LIN {X 0,Y 421.237,Z 718.592,A -85,B 0,C 180,E1 -10154.642,E2 -10154.642} C_VEL
LIN {X 0,Y 420.431,Z 729.964,A -85,B 0,C 180,E1 -10155.589,E2 -10155.589} C_VEL
LIN {X 0,Y 419.711,Z 740.495,A -85,B 0,C 180,E1 -10156.689,E2 -10156.689} C_VEL
LIN {X 0,Y 419.004,Z 749.849,A -85,B 0,C 180,E1 -10157.898,E2 -10157.898} C_VEL
LIN {X 0,Y 418.229,Z 758.896,A -85,B 0,C 180,E1 -10159.348,E2 -10159.348} C_VEL
LIN {X 0,Y 417.744,Z 766.199,A -85,B 0,C 180,E1 -10160.803,E2 -10160.803} C_VEL
LIN {X 0,Y 417.402,Z 772.062,A -85,B 0,C 180,E1 -10162.259,E2 -10162.259} C_VEL
LIN {X 0,Y 417.147,Z 776.738,A -85,B 0,C 180,E1 -10163.731,E2 -10163.731} C_VEL
LIN {X 0,Y 417.113,Z 780.212,A -85,B 0,C 180,E1 -10165.167,E2 -10165.167} C_VEL
LIN {X 0,Y 417.016,Z 782.003,A -85,B 0,C 180,E1 -10166.135,E2 -10166.135} C_VEL
LIN {X 0,Y 417.028,Z 783.359,A -85,B 0,C 180,E1 -10167.102,E2 -10167.102} C_VEL
LIN {X 0,Y 417.056,Z 784.323,A -85,B 0,C 180,E1 -10168.069,E2 -10168.069} C_VEL
LIN {X 0,Y 417.01,Z 784.898,A -85,B 0,C 180,E1 -10169.034,E2 -10169.034} C_VEL
LIN {X 0,Y 417.003,Z 785.053,A -85,B 0,C 180,E1 -10170,E2 -10170} C_VEL
LIN {X 0,Y 417.056,Z 784.159,A -85,B 0,C 180,E1 -10171.931,E2 -10171.931} C_VEL
LIN {X 0,Y 417.03,Z 783.127,A -85,B 0,C 180,E1 -10172.898,E2 -10172.898} C_VEL
LIN {X 0,Y 417.017,Z 781.664,A -85,B 0,C 180,E1 -10173.865,E2 -10173.865} C_VEL
LIN {X 0,Y 417.131,Z 778.661,A -85,B 0,C 180,E1 -10175.317,E2 -10175.317} C_VEL
LIN {X 0,Y 417.234,Z 774.598,A -85,B 0,C 180,E1 -10176.771,E2 -10176.771} C_VEL
LIN {X 0,Y 417.539,Z 768.351,A -85,B 0,C 180,E1 -10178.469,E2 -10178.469} C_VEL
LIN {X 0,Y 417.941,Z 761.546,A -85,B 0,C 180,E1 -10179.925,E2 -10179.925} C_VEL
LIN {X 0,Y 418.494,Z 753.083,A -85,B 0,C 180,E1 -10181.38,E2 -10181.38} C_VEL
LIN {X 0,Y 419.161,Z 744.361,A -85,B 0,C 180,E1 -10182.589,E2 -10182.589} C_VEL
LIN {X 0,Y 419.889,Z 733.598,A -85,B 0,C 180,E1 -10183.8,E2 -10183.8} C_VEL
LIN {X 0,Y 420.541,Z 722.919,A -85,B 0,C 180,E1 -10184.765,E2 -10184.765} C_VEL
LIN {X 0,Y 421.282,Z 710.937,A -85,B 0,C 180,E1 -10185.605,E2 -10185.605} C_VEL
LIN {X 0,Y 421.895,Z 698.447,A -85,B 0,C 180,E1 -10186.264,E2 -10186.264} C_VEL
LIN {X 0,Y 422.437,Z 685.494,A -85,B 0,C 180,E1 -10186.739,E2 -10186.739} C_VEL
LIN {X 0,Y 422.751,Z 669.81,A -85,B 0,C 180,E1 -10187.069,E2 -10187.069} C_VEL
LIN {X 0,Y 423.344,Z 596.874,A -85,B 0,C 180,E1 -10188.309,E2 -10188.309} C_VEL
LIN {X 0,Y 419.621,Z 572.484,A -85,B 0,C 180,E1 -10188.908,E2 -10188.908} C_VEL
LIN {X 0,Y 420.653,Z 555.298,A -85,B 0,C 180,E1 -10192.339,E2 -10192.339} C_VEL
LIN {X 0,Y 421.132,Z 547.688,A -85,B 0,C 180,E1 -10193.871,E2 -10193.871} C_VEL
LIN {X 0,Y 419.064,Z 536.126,A -85,B 0,C 180,E1 -10196.386,E2 -10196.386} C_VEL
LIN {X 0,Y 418.336,Z 532.377,A -85,B 0,C 180,E1 -10197.246,E2 -10197.246} C_VEL
LIN {X 0,Y 418.244,Z 532.387,A -85,B 0,C 180,E1 -10200.271,E2 -10200.271} C_VEL
LIN {X 0,Y 418.247,Z 532.387,A -85,B 0,C 180,E1 -10203.676,E2 -10203.676} C_VEL
LIN {X 0,Y 418.243,Z 532.387,A -85,B 0,C 180,E1 -10207.223,E2 -10207.223} C_VEL
LIN {X 0,Y 418.252,Z 532.386,A -85,B 0,C 180,E1 -10209.681,E2 -10209.681} C_VEL
LIN {X 0,Y 418.228,Z 532.384,A -85,B 0,C 180,E1 -10212.321,E2 -10212.321} C_VEL
LIN {X 0,Y 418.234,Z 532.387,A -85,B 0,C 180,E1 -10215.108,E2 -10215.108} C_VEL
LIN {X 0,Y 418.251,Z 532.385,A -85,B 0,C 180,E1 -10217.768,E2 -10217.768} C_VEL
LIN {X 0,Y 418.263,Z 532.38,A -85,B 0,C 180,E1 -10220.616,E2 -10220.616} C_VEL
LIN {X 0,Y 418.24,Z 532.385,A -85,B 0,C 180,E1 -10223.975,E2 -10223.975} C_VEL
LIN {X 0,Y 418.251,Z 532.385,A -85,B 0,C 180,E1 -10227.155,E2 -10227.155} C_VEL
LIN {X 0,Y 418.267,Z 532.381,A -85,B 0,C 180,E1 -10230.838,E2 -10230.838} C_VEL
LIN {X 0,Y 418.263,Z 532.381,A -85,B 0,C 180,E1 -10234.095,E2 -10234.095} C_VEL
LIN {X 0,Y 418.224,Z 532.39,A -85,B 0,C 180,E1 -10237.263,E2 -10237.263} C_VEL
LIN {X 0,Y 418.275,Z 532.379,A -85,B 0,C 180,E1 -10240.364,E2 -10240.364} C_VEL
LIN {X 0,Y 418.308,Z 532.382,A -85,B 0,C 180,E1 -10243.404,E2 -10243.404} C_VEL
LIN {X 0,Y 418.337,Z 532.373,A -85,B 0,C 180,E1 -10246.999,E2 -10246.999} C_VEL
LIN {X 0,Y 418.333,Z 532.371,A -85,B 0,C 180,E1 -10250.329,E2 -10250.329} C_VEL
LIN {X 0,Y 418.484,Z 532.358,A -85,B 0,C 180,E1 -10253.249,E2 -10253.249} C_VEL
LIN {X 0,Y 418.333,Z 532.376,A -85,B 0,C 180,E1 -10255.182,E2 -10255.182} C_VEL
LIN {X 0,Y 418.536,Z 532.347,A -85,B 0,C 180,E1 -10258.076,E2 -10258.076} C_VEL
LIN {X 0,Y 418.663,Z 532.332,A -85,B 0,C 180,E1 -10260,E2 -10260} C_VEL
LIN {X 0,Y 418.503,Z 532.352,A -85,B 0,C 180,E1 -10262.888,E2 -10262.888} C_VEL
LIN {X 0,Y 418.486,Z 532.353,A -85,B 0,C 180,E1 -10266.751,E2 -10266.751} C_VEL
LIN {X 0,Y 418.333,Z 532.376,A -85,B 0,C 180,E1 -10269.672,E2 -10269.672} C_VEL
LIN {X 0,Y 418.338,Z 532.373,A -85,B 0,C 180,E1 -10273.001,E2 -10273.001} C_VEL
LIN {X 0,Y 418.305,Z 532.376,A -85,B 0,C 180,E1 -10276.736,E2 -10276.736} C_VEL
LIN {X 0,Y 418.263,Z 532.383,A -85,B 0,C 180,E1 -10279.791,E2 -10279.791} C_VEL
LIN {X 0,Y 418.231,Z 532.385,A -85,B 0,C 180,E1 -10282.737,E2 -10282.737} C_VEL
LIN {X 0,Y 418.265,Z 532.382,A -85,B 0,C 180,E1 -10285.905,E2 -10285.905} C_VEL
LIN {X 0,Y 418.269,Z 532.384,A -85,B 0,C 180,E1 -10289.162,E2 -10289.162} C_VEL
LIN {X 0,Y 418.252,Z 532.383,A -85,B 0,C 180,E1 -10292.845,E2 -10292.845} C_VEL
LIN {X 0,Y 418.243,Z 532.383,A -85,B 0,C 180,E1 -10296.239,E2 -10296.239} C_VEL
LIN {X 0,Y 418.251,Z 532.386,A -85,B 0,C 180,E1 -10299.682,E2 -10299.682} C_VEL
LIN {X 0,Y 418.228,Z 532.384,A -85,B 0,C 180,E1 -10302.322,E2 -10302.322} C_VEL
LIN {X 0,Y 418.258,Z 532.385,A -85,B 0,C 180,E1 -10305.113,E2 -10305.113} C_VEL
LIN {X 0,Y 418.29,Z 532.38,A -85,B 0,C 180,E1 -10307.774,E2 -10307.774} C_VEL
LIN {X 0,Y 418.265,Z 532.385,A -85,B 0,C 180,E1 -10311.561,E2 -10311.561} C_VEL
LIN {X 0,Y 418.259,Z 532.385,A -85,B 0,C 180,E1 -10315.16,E2 -10315.16} C_VEL
LIN {X 0,Y 418.245,Z 532.389,A -85,B 0,C 180,E1 -10317.473,E2 -10317.473} C_VEL
LIN {X 0,Y 418.269,Z 532.381,A -85,B 0,C 180,E1 -10320.896,E2 -10320.896} C_VEL
LIN {X 0,Y 418.272,Z 532.38,A -85,B 0,C 180,E1 -10324.097,E2 -10324.097} C_VEL
LIN {X 0,Y 418.24,Z 532.389,A -85,B 0,C 180,E1 -10327.265,E2 -10327.265} C_VEL
LIN {X 0,Y 418.339,Z 532.468,A -85,B 0,C 180,E1 -10330.782,E2 -10330.782} C_VEL
LIN {X 0,Y 420.02,Z 541.497,A -85,B 0,C 180,E1 -10333.063,E2 -10333.063} C_VEL
LIN {X 0,Y 420.061,Z 546.37,A -85,B 0,C 180,E1 -10334.224,E2 -10334.224} C_VEL
LIN {X 0,Y 419.823,Z 550.579,A -85,B 0,C 180,E1 -10335.189,E2 -10335.189} C_VEL
LIN {X 0,Y 423.668,Z 570.868,A -85,B 0,C 180,E1 -10335.708,E2 -10335.708} C_VEL
LIN {X 0,Y 422.734,Z 656.919,A -85,B 0,C 180,E1 -10337.183,E2 -10337.183} C_VEL
LIN {X 0,Y 422.345,Z 670.234,A -85,B 0,C 180,E1 -10337.599,E2 -10337.599} C_VEL
LIN {X 0,Y 421.806,Z 683.503,A -85,B 0,C 180,E1 -10338.223,E2 -10338.223} C_VEL
LIN {X 0,Y 421.245,Z 694.646,A -85,B 0,C 180,E1 -10338.939,E2 -10338.939} C_VEL
LIN {X 0,Y 420.556,Z 706.179,A -85,B 0,C 180,E1 -10339.894,E2 -10339.894} C_VEL
LIN {X 0,Y 419.728,Z 716.568,A -85,B 0,C 180,E1 -10340.969,E2 -10340.969} C_VEL
LIN {X 0,Y 419.154,Z 725.534,A -85,B 0,C 180,E1 -10342.115,E2 -10342.115} C_VEL
LIN {X 0,Y 418.647,Z 734.156,A -85,B 0,C 180,E1 -10343.477,E2 -10343.477} C_VEL
LIN {X 0,Y 417.73,Z 737.728,A -85,B 0,C 180,E1 -10344.111,E2 -10344.111} C_VEL
LIN {X 0,Y 414.518,Z 743.104,A -85,B 0,C 180,E1 -10345.171,E2 -10345.171} C_VEL
LIN {X 0,Y 411.29,Z 747.831,A -85,B 0,C 180,E1 -10346.299,E2 -10346.299} C_VEL
LIN {X 0,Y 410.362,Z 750.362,A -85,B 0,C 180,E1 -10347.032,E2 -10347.032} C_VEL
LIN {X 0,Y 410.196,Z 754.534,A -85,B 0,C 180,E1 -10348.527,E2 -10348.527} C_VEL
LIN {X 0,Y 409.964,Z 757.597,A -85,B 0,C 180,E1 -10350,E2 -10350} C_VEL
LIN {X 0,Y 409.959,Z 759.12,A -85,B 0,C 180,E1 -10350.982,E2 -10350.982} C_VEL
LIN {X 0,Y 410.004,Z 760.199,A -85,B 0,C 180,E1 -10351.965,E2 -10351.965} C_VEL
LIN {X 0,Y 409.905,Z 761.188,A -85,B 0,C 180,E1 -10353.932,E2 -10353.932} C_VEL
LIN {X 0,Y 409.962,Z 761.111,A -85,B 0,C 180,E1 -10354.917,E2 -10354.917} C_VEL
LIN {X 0,Y 410.006,Z 760.392,A -85,B 0,C 180,E1 -10356.175,E2 -10356.175} C_VEL
LIN {X 0,Y 410.055,Z 758.414,A -85,B 0,C 180,E1 -10357.881,E2 -10357.881} C_VEL
LIN {X 0,Y 410.171,Z 755.664,A -85,B 0,C 180,E1 -10359.368,E2 -10359.368} C_VEL
LIN {X 0,Y 410.443,Z 751.886,A -85,B 0,C 180,E1 -10360.856,E2 -10360.856} C_VEL
LIN {X 0,Y 410.773,Z 746.972,A -85,B 0,C 180,E1 -10362.349,E2 -10362.349} C_VEL
LIN {X 0,Y 411.238,Z 740.769,A -85,B 0,C 180,E1 -10363.842,E2 -10363.842} C_VEL
LIN {X 0,Y 411.926,Z 733.001,A -85,B 0,C 180,E1 -10365.334,E2 -10365.334} C_VEL
LIN {X 0,Y 412.653,Z 725.035,A -85,B 0,C 180,E1 -10366.575,E2 -10366.575} C_VEL
LIN {X 0,Y 413.383,Z 715.288,A -85,B 0,C 180,E1 -10367.819,E2 -10367.819} C_VEL
LIN {X 0,Y 414.224,Z 704.42,A -85,B 0,C 180,E1 -10368.934,E2 -10368.934} C_VEL
LIN {X 0,Y 414.998,Z 693.767,A -85,B 0,C 180,E1 -10369.797,E2 -10369.797} C_VEL
LIN {X 0,Y 415.777,Z 680.905,A -85,B 0,C 180,E1 -10370.597,E2 -10370.597} C_VEL
LIN {X 0,Y 416.286,Z 668.677,A -85,B 0,C 180,E1 -10371.153,E2 -10371.153} C_VEL
LIN {X 0,Y 416.656,Z 656.324,A -85,B 0,C 180,E1 -10371.522,E2 -10371.522} C_VEL
LIN {X 0,Y 417.668,Z 571.191,A -85,B 0,C 180,E1 -10373.014,E2 -10373.014} C_VEL
LIN {X 0,Y 413.325,Z 550.756,A -85,B 0,C 180,E1 -10373.626,E2 -10373.626} C_VEL
LIN {X 0,Y 413.542,Z 545.618,A -85,B 0,C 180,E1 -10374.873,E2 -10374.873} C_VEL
LIN {X 0,Y 411.819,Z 535.822,A -85,B 0,C 180,E1 -10377.436,E2 -10377.436} C_VEL
LIN {X 0,Y 411.258,Z 533.253,A -85,B 0,C 180,E1 -10378.169,E2 -10378.169} C_VEL
LIN {X 0,Y 411.183,Z 533.263,A -85,B 0,C 180,E1 -10381.283,E2 -10381.283} C_VEL
LIN {X 0,Y 411.206,Z 533.266,A -85,B 0,C 180,E1 -10384.333,E2 -10384.333} C_VEL
LIN {X 0,Y 411.203,Z 533.26,A -85,B 0,C 180,E1 -10387.972,E2 -10387.972} C_VEL
LIN {X 0,Y 411.208,Z 533.261,A -85,B 0,C 180,E1 -10391.235,E2 -10391.235} C_VEL
LIN {X 0,Y 411.223,Z 533.263,A -85,B 0,C 180,E1 -10394.483,E2 -10394.483} C_VEL
LIN {X 0,Y 411.196,Z 533.261,A -85,B 0,C 180,E1 -10398.196,E2 -10398.196} C_VEL
LIN {X 0,Y 411.223,Z 533.262,A -85,B 0,C 180,E1 -10400.776,E2 -10400.776} C_VEL
LIN {X 0,Y 411.195,Z 533.266,A -85,B 0,C 180,E1 -10404.471,E2 -10404.471} C_VEL
LIN {X 0,Y 411.163,Z 533.267,A -85,B 0,C 180,E1 -10408.002,E2 -10408.002} C_VEL
LIN {X 0,Y 411.218,Z 533.259,A -85,B 0,C 180,E1 -10411.41,E2 -10411.41} C_VEL
LIN {X 0,Y 411.23,Z 533.261,A -85,B 0,C 180,E1 -10414.706,E2 -10414.706} C_VEL
LIN {X 0,Y 411.198,Z 533.256,A -85,B 0,C 180,E1 -10417.913,E2 -10417.913} C_VEL
LIN {X 0,Y 411.216,Z 533.258,A -85,B 0,C 180,E1 -10421.051,E2 -10421.051} C_VEL
LIN {X 0,Y 411.246,Z 533.256,A -85,B 0,C 180,E1 -10424.131,E2 -10424.131} C_VEL
LIN {X 0,Y 411.294,Z 533.245,A -85,B 0,C 180,E1 -10427.165,E2 -10427.165} C_VEL
LIN {X 0,Y 411.285,Z 533.252,A -85,B 0,C 180,E1 -10430.161,E2 -10430.161} C_VEL
LIN {X 0,Y 411.448,Z 533.229,A -85,B 0,C 180,E1 -10433.133,E2 -10433.133} C_VEL
LIN {X 0,Y 411.305,Z 533.25,A -85,B 0,C 180,E1 -10435.099,E2 -10435.099} C_VEL
LIN {X 0,Y 411.505,Z 533.218,A -85,B 0,C 180,E1 -10438.042,E2 -10438.042} C_VEL
LIN {X 0,Y 411.634,Z 533.207,A -85,B 0,C 180,E1 -10440,E2 -10440} C_VEL
LIN {X 0,Y 411.458,Z 533.226,A -85,B 0,C 180,E1 -10442.937,E2 -10442.937} C_VEL
LIN {X 0,Y 411.447,Z 533.231,A -85,B 0,C 180,E1 -10446.867,E2 -10446.867} C_VEL
LIN {X 0,Y 411.285,Z 533.248,A -85,B 0,C 180,E1 -10449.839,E2 -10449.839} C_VEL
LIN {X 0,Y 411.297,Z 533.244,A -85,B 0,C 180,E1 -10453.104,E2 -10453.104} C_VEL
LIN {X 0,Y 411.255,Z 533.256,A -85,B 0,C 180,E1 -10456.869,E2 -10456.869} C_VEL
LIN {X 0,Y 411.222,Z 533.258,A -85,B 0,C 180,E1 -10459.987,E2 -10459.987} C_VEL
LIN {X 0,Y 411.189,Z 533.26,A -85,B 0,C 180,E1 -10463.148,E2 -10463.148} C_VEL
LIN {X 0,Y 411.231,Z 533.261,A -85,B 0,C 180,E1 -10466.381,E2 -10466.381} C_VEL
LIN {X 0,Y 411.204,Z 533.26,A -85,B 0,C 180,E1 -10469.712,E2 -10469.712} C_VEL
LIN {X 0,Y 411.2,Z 533.262,A -85,B 0,C 180,E1 -10473.156,E2 -10473.156} C_VEL
LIN {X 0,Y 411.19,Z 533.268,A -85,B 0,C 180,E1 -10476.554,E2 -10476.554} C_VEL
LIN {X 0,Y 411.222,Z 533.258,A -85,B 0,C 180,E1 -10479.731,E2 -10479.731} C_VEL
LIN {X 0,Y 411.172,Z 533.267,A -85,B 0,C 180,E1 -10483.134,E2 -10483.134} C_VEL
LIN {X 0,Y 411.169,Z 533.266,A -85,B 0,C 180,E1 -10485.881,E2 -10485.881} C_VEL
LIN {X 0,Y 411.163,Z 533.271,A -85,B 0,C 180,E1 -10488.772,E2 -10488.772} C_VEL
LIN {X 0,Y 411.208,Z 533.262,A -85,B 0,C 180,E1 -10491.831,E2 -10491.831} C_VEL
LIN {X 0,Y 411.209,Z 533.263,A -85,B 0,C 180,E1 -10495.122,E2 -10495.122} C_VEL
LIN {X 0,Y 411.164,Z 533.27,A -85,B 0,C 180,E1 -10498.004,E2 -10498.004} C_VEL
LIN {X 0,Y 411.265,Z 533.257,A -85,B 0,C 180,E1 -10501.832,E2 -10501.832} C_VEL
LIN {X 0,Y 411.322,Z 533.527,A -85,B 0,C 180,E1 -10501.975,E2 -10501.975} C_VEL
LIN {X 0,Y 413.922,Z 545.976,A -85,B 0,C 180,E1 -10504.883,E2 -10504.883} C_VEL
LIN {X 0,Y 414.629,Z 550.956,A -85,B 0,C 180,E1 -10505.997,E2 -10505.997} C_VEL
LIN {X 0,Y 413.433,Z 565.861,A -85,B 0,C 180,E1 -10509.086,E2 -10509.086} C_VEL
LIN {X 0,Y 413.028,Z 572.239,A -85,B 0,C 180,E1 -10510.398,E2 -10510.398} C_VEL
LIN {X 0,Y 416.99,Z 595.24,A -85,B 0,C 180,E1 -10511.027,E2 -10511.027} C_VEL
LIN {X 0,Y 417.461,Z 600.988,A -85,B 0,C 180,E1 -10511.154,E2 -10511.154} C_VEL
LIN {X 0,Y 416.494,Z 679.959,A -85,B 0,C 180,E1 -10512.54,E2 -10512.54} C_VEL
LIN {X 0,Y 415.926,Z 693.364,A -85,B 0,C 180,E1 -10512.959,E2 -10512.959} C_VEL
LIN {X 0,Y 415.382,Z 704.447,A -85,B 0,C 180,E1 -10513.474,E2 -10513.474} C_VEL
LIN {X 0,Y 414.53,Z 717.067,A -85,B 0,C 180,E1 -10514.261,E2 -10514.261} C_VEL
LIN {X 0,Y 413.646,Z 728.858,A -85,B 0,C 180,E1 -10515.235,E2 -10515.235} C_VEL
LIN {X 0,Y 412.81,Z 739.421,A -85,B 0,C 180,E1 -10516.337,E2 -10516.337} C_VEL
LIN {X 0,Y 412.172,Z 748.063,A -85,B 0,C 180,E1 -10517.444,E2 -10517.444} C_VEL
LIN {X 0,Y 411.465,Z 756.034,A -85,B 0,C 180,E1 -10518.672,E2 -10518.672} C_VEL
LIN {X 0,Y 410.87,Z 763.857,A -85,B 0,C 180,E1 -10520.151,E2 -10520.151} C_VEL
LIN {X 0,Y 410.466,Z 770.122,A -85,B 0,C 180,E1 -10521.632,E2 -10521.632} C_VEL
LIN {X 0,Y 410.169,Z 775.115,A -85,B 0,C 180,E1 -10523.111,E2 -10523.111} C_VEL
LIN {X 0,Y 410.028,Z 778.983,A -85,B 0,C 180,E1 -10524.591,E2 -10524.591} C_VEL
LIN {X 0,Y 409.935,Z 781.83,A -85,B 0,C 180,E1 -10526.068,E2 -10526.068} C_VEL
LIN {X 0,Y 409.966,Z 784.137,A -85,B 0,C 180,E1 -10528.035,E2 -10528.035} C_VEL
LIN {X 0,Y 409.935,Z 784.704,A -85,B 0,C 180,E1 -10529.018,E2 -10529.018} C_VEL
LIN {X 0,Y 409.926,Z 784.846,A -85,B 0,C 180,E1 -10530,E2 -10530} C_VEL
LIN {X 0,Y 409.967,Z 783.936,A -85,B 0,C 180,E1 -10531.965,E2 -10531.965} C_VEL
LIN {X 0,Y 409.928,Z 782.897,A -85,B 0,C 180,E1 -10532.948,E2 -10532.948} C_VEL
LIN {X 0,Y 409.935,Z 781.419,A -85,B 0,C 180,E1 -10533.932,E2 -10533.932} C_VEL
LIN {X 0,Y 410.027,Z 778.401,A -85,B 0,C 180,E1 -10535.409,E2 -10535.409} C_VEL
LIN {X 0,Y 410.167,Z 774.321,A -85,B 0,C 180,E1 -10536.889,E2 -10536.889} C_VEL
LIN {X 0,Y 410.488,Z 768.054,A -85,B 0,C 180,E1 -10538.616,E2 -10538.616} C_VEL
LIN {X 0,Y 410.924,Z 761.228,A -85,B 0,C 180,E1 -10540.096,E2 -10540.096} C_VEL
LIN {X 0,Y 411.51,Z 752.727,A -85,B 0,C 180,E1 -10541.576,E2 -10541.576} C_VEL
LIN {X 0,Y 412.2,Z 743.974,A -85,B 0,C 180,E1 -10542.806,E2 -10542.806} C_VEL
LIN {X 0,Y 412.952,Z 733.04,A -85,B 0,C 180,E1 -10544.051,E2 -10544.051} C_VEL
LIN {X 0,Y 413.646,Z 722.433,A -85,B 0,C 180,E1 -10545.016,E2 -10545.016} C_VEL
LIN {X 0,Y 414.428,Z 710.356,A -85,B 0,C 180,E1 -10545.869,E2 -10545.869} C_VEL
LIN {X 0,Y 415.066,Z 697.749,A -85,B 0,C 180,E1 -10546.539,E2 -10546.539} C_VEL
LIN {X 0,Y 415.605,Z 685.545,A -85,B 0,C 180,E1 -10546.991,E2 -10546.991} C_VEL
LIN {X 0,Y 415.909,Z 671.838,A -85,B 0,C 180,E1 -10547.295,E2 -10547.295} C_VEL
LIN {X 0,Y 416.582,Z 597.736,A -85,B 0,C 180,E1 -10548.573,E2 -10548.573} C_VEL
LIN {X 0,Y 412.651,Z 572.33,A -85,B 0,C 180,E1 -10549.203,E2 -10549.203} C_VEL
LIN {X 0,Y 413.813,Z 554.98,A -85,B 0,C 180,E1 -10552.729,E2 -10552.729} C_VEL
LIN {X 0,Y 414.155,Z 548.636,A -85,B 0,C 180,E1 -10554.033,E2 -10554.033} C_VEL
LIN {X 0,Y 412.041,Z 537.078,A -85,B 0,C 180,E1 -10556.598,E2 -10556.598} C_VEL
LIN {X 0,Y 411.286,Z 533.256,A -85,B 0,C 180,E1 -10557.475,E2 -10557.475} C_VEL
LIN {X 0,Y 411.188,Z 533.267,A -85,B 0,C 180,E1 -10560.847,E2 -10560.847} C_VEL
LIN {X 0,Y 411.204,Z 533.26,A -85,B 0,C 180,E1 -10564.333,E2 -10564.333} C_VEL
LIN {X 0,Y 411.198,Z 533.262,A -85,B 0,C 180,E1 -10567.972,E2 -10567.972} C_VEL
LIN {X 0,Y 411.18,Z 533.262,A -85,B 0,C 180,E1 -10570.503,E2 -10570.503} C_VEL
LIN {X 0,Y 411.174,Z 533.266,A -85,B 0,C 180,E1 -10573.132,E2 -10573.132} C_VEL
LIN {X 0,Y 411.164,Z 533.267,A -85,B 0,C 180,E1 -10575.88,E2 -10575.88} C_VEL
LIN {X 0,Y 411.195,Z 533.261,A -85,B 0,C 180,E1 -10578.765,E2 -10578.765} C_VEL
LIN {X 0,Y 411.199,Z 533.261,A -85,B 0,C 180,E1 -10582.027,E2 -10582.027} C_VEL
LIN {X 0,Y 411.2,Z 533.265,A -85,B 0,C 180,E1 -10585.666,E2 -10585.666} C_VEL
LIN {X 0,Y 411.191,Z 533.265,A -85,B 0,C 180,E1 -10589.153,E2 -10589.153} C_VEL
LIN {X 0,Y 411.253,Z 533.253,A -85,B 0,C 180,E1 -10592.522,E2 -10592.522} C_VEL
LIN {X 0,Y 411.213,Z 533.262,A -85,B 0,C 180,E1 -10595.784,E2 -10595.784} C_VEL
LIN {X 0,Y 411.188,Z 533.263,A -85,B 0,C 180,E1 -10598.965,E2 -10598.965} C_VEL
LIN {X 0,Y 411.244,Z 533.255,A -85,B 0,C 180,E1 -10602.085,E2 -10602.085} C_VEL
LIN {X 0,Y 411.252,Z 533.257,A -85,B 0,C 180,E1 -10605.147,E2 -10605.147} C_VEL
LIN {X 0,Y 411.276,Z 533.251,A -85,B 0,C 180,E1 -10608.167,E2 -10608.167} C_VEL
LIN {X 0,Y 411.434,Z 533.231,A -85,B 0,C 180,E1 -10612.186,E2 -10612.186} C_VEL
LIN {X 0,Y 411.466,Z 533.227,A -85,B 0,C 180,E1 -10614.118,E2 -10614.118} C_VEL
LIN {X 0,Y 411.505,Z 533.223,A -85,B 0,C 180,E1 -10618.043,E2 -10618.043} C_VEL
LIN {X 0,Y 411.632,Z 533.207,A -85,B 0,C 180,E1 -10620,E2 -10620} C_VEL
LIN {X 0,Y 411.459,Z 533.23,A -85,B 0,C 180,E1 -10622.937,E2 -10622.937} C_VEL
LIN {X 0,Y 411.443,Z 533.23,A -85,B 0,C 180,E1 -10626.646,E2 -10626.646} C_VEL
LIN {X 0,Y 411.285,Z 533.252,A -85,B 0,C 180,E1 -10629.839,E2 -10629.839} C_VEL
LIN {X 0,Y 411.297,Z 533.251,A -85,B 0,C 180,E1 -10633.104,E2 -10633.104} C_VEL
LIN {X 0,Y 411.255,Z 533.255,A -85,B 0,C 180,E1 -10636.869,E2 -10636.869} C_VEL
LIN {X 0,Y 411.223,Z 533.258,A -85,B 0,C 180,E1 -10639.987,E2 -10639.987} C_VEL
LIN {X 0,Y 411.196,Z 533.264,A -85,B 0,C 180,E1 -10643.148,E2 -10643.148} C_VEL
LIN {X 0,Y 411.232,Z 533.256,A -85,B 0,C 180,E1 -10646.382,E2 -10646.382} C_VEL
LIN {X 0,Y 411.205,Z 533.263,A -85,B 0,C 180,E1 -10649.713,E2 -10649.713} C_VEL
LIN {X 0,Y 411.201,Z 533.264,A -85,B 0,C 180,E1 -10653.157,E2 -10653.157} C_VEL
LIN {X 0,Y 411.191,Z 533.261,A -85,B 0,C 180,E1 -10656.554,E2 -10656.554} C_VEL
LIN {X 0,Y 411.214,Z 533.262,A -85,B 0,C 180,E1 -10659.73,E2 -10659.73} C_VEL
LIN {X 0,Y 411.175,Z 533.267,A -85,B 0,C 180,E1 -10663.134,E2 -10663.134} C_VEL
LIN {X 0,Y 411.225,Z 533.259,A -85,B 0,C 180,E1 -10665.873,E2 -10665.873} C_VEL
LIN {X 0,Y 411.208,Z 533.26,A -85,B 0,C 180,E1 -10668.765,E2 -10668.765} C_VEL
LIN {X 0,Y 411.203,Z 533.26,A -85,B 0,C 180,E1 -10672.028,E2 -10672.028} C_VEL
LIN {X 0,Y 411.206,Z 533.263,A -85,B 0,C 180,E1 -10675.667,E2 -10675.667} C_VEL
LIN {X 0,Y 411.19,Z 533.266,A -85,B 0,C 180,E1 -10679.153,E2 -10679.153} C_VEL
LIN {X 0,Y 411.26,Z 533.253,A -85,B 0,C 180,E1 -10682.523,E2 -10682.523} C_VEL
LIN {X 0,Y 411.229,Z 533.259,A -85,B 0,C 180,E1 -10685.785,E2 -10685.785} C_VEL
LIN {X 0,Y 411.199,Z 533.269,A -85,B 0,C 180,E1 -10688.967,E2 -10688.967} C_VEL
LIN {X 0,Y 411.28,Z 533.366,A -85,B 0,C 180,E1 -10690.569,E2 -10690.569} C_VEL
LIN {X 0,Y 413.157,Z 543.6,A -85,B 0,C 180,E1 -10693.192,E2 -10693.192} C_VEL
LIN {X 0,Y 412.914,Z 550.674,A -85,B 0,C 180,E1 -10694.879,E2 -10694.879} C_VEL
LIN {X 0,Y 416.89,Z 571.558,A -85,B 0,C 180,E1 -10695.432,E2 -10695.432} C_VEL
LIN {X 0,Y 415.916,Z 657.716,A -85,B 0,C 180,E1 -10696.938,E2 -10696.938} C_VEL
LIN {X 0,Y 415.484,Z 670.83,A -85,B 0,C 180,E1 -10697.359,E2 -10697.359} C_VEL
LIN {X 0,Y 414.951,Z 683.439,A -85,B 0,C 180,E1 -10697.964,E2 -10697.964} C_VEL
LIN {X 0,Y 414.338,Z 695.446,A -85,B 0,C 180,E1 -10698.752,E2 -10698.752} C_VEL
LIN {X 0,Y 413.619,Z 706.871,A -85,B 0,C 180,E1 -10699.723,E2 -10699.723} C_VEL
LIN {X 0,Y 412.749,Z 717.178,A -85,B 0,C 180,E1 -10700.815,E2 -10700.815} C_VEL
LIN {X 0,Y 412.157,Z 726.127,A -85,B 0,C 180,E1 -10701.99,E2 -10701.99} C_VEL
LIN {X 0,Y 411.596,Z 734.717,A -85,B 0,C 180,E1 -10703.382,E2 -10703.382} C_VEL
LIN {X 0,Y 411.062,Z 742.059,A -85,B 0,C 180,E1 -10704.85,E2 -10704.85} C_VEL
LIN {X 0,Y 410.557,Z 748.832,A -85,B 0,C 180,E1 -10706.565,E2 -10706.565} C_VEL
LIN {X 0,Y 410.362,Z 750.362,A -85,B 0,C 180,E1 -10707.032,E2 -10707.032} C_VEL
LIN {X 0,Y 409.471,Z 752.708,A -85,B 0,C 180,E1 -10707.781,E2 -10707.781} C_VEL
LIN {X 0,Y 406.442,Z 756.002,A -85,B 0,C 180,E1 -10709.025,E2 -10709.025} C_VEL
LIN {X 0,Y 404.002,Z 758.049,A -85,B 0,C 180,E1 -10710.055,E2 -10710.055} C_VEL
LIN {X 0,Y 402.966,Z 759.224,A -85,B 0,C 180,E1 -10710.866,E2 -10710.866} C_VEL
LIN {X 0,Y 402.882,Z 759.538,A -85,B 0,C 180,E1 -10711.143,E2 -10711.143} C_VEL
LIN {X 0,Y 402.914,Z 760.441,A -85,B 0,C 180,E1 -10711.999,E2 -10711.999} C_VEL
LIN {X 0,Y 402.824,Z 761.4,A -85,B 0,C 180,E1 -10714.002,E2 -10714.002} C_VEL
LIN {X 0,Y 402.875,Z 761.304,A -85,B 0,C 180,E1 -10715.004,E2 -10715.004} C_VEL
LIN {X 0,Y 402.933,Z 760.648,A -85,B 0,C 180,E1 -10716.171,E2 -10716.171} C_VEL
LIN {X 0,Y 402.981,Z 758.55,A -85,B 0,C 180,E1 -10718.02,E2 -10718.02} C_VEL
LIN {X 0,Y 403.107,Z 755.769,A -85,B 0,C 180,E1 -10719.534,E2 -10719.534} C_VEL
LIN {X 0,Y 403.429,Z 751.957,A -85,B 0,C 180,E1 -10721.047,E2 -10721.047} C_VEL
LIN {X 0,Y 403.745,Z 747.201,A -85,B 0,C 180,E1 -10722.512,E2 -10722.512} C_VEL
LIN {X 0,Y 404.277,Z 740.763,A -85,B 0,C 180,E1 -10724.086,E2 -10724.086} C_VEL
LIN {X 0,Y 404.997,Z 732.925,A -85,B 0,C 180,E1 -10725.603,E2 -10725.603} C_VEL
LIN {X 0,Y 405.793,Z 724.904,A -85,B 0,C 180,E1 -10726.863,E2 -10726.863} C_VEL
LIN {X 0,Y 406.577,Z 715.091,A -85,B 0,C 180,E1 -10728.128,E2 -10728.128} C_VEL
LIN {X 0,Y 407.45,Z 704.109,A -85,B 0,C 180,E1 -10729.261,E2 -10729.261} C_VEL
LIN {X 0,Y 408.259,Z 693.309,A -85,B 0,C 180,E1 -10730.138,E2 -10730.138} C_VEL
LIN {X 0,Y 409.068,Z 680.262,A -85,B 0,C 180,E1 -10730.95,E2 -10730.95} C_VEL
LIN {X 0,Y 409.597,Z 668.498,A -85,B 0,C 180,E1 -10731.482,E2 -10731.482} C_VEL
LIN {X 0,Y 409.974,Z 655.79,A -85,B 0,C 180,E1 -10731.858,E2 -10731.858} C_VEL
LIN {X 0,Y 411.056,Z 572.3,A -85,B 0,C 180,E1 -10733.341,E2 -10733.341} C_VEL
LIN {X 0,Y 406.484,Z 550.932,A -85,B 0,C 180,E1 -10734.003,E2 -10734.003} C_VEL
LIN {X 0,Y 406.596,Z 546.69,A -85,B 0,C 180,E1 -10735.054,E2 -10735.054} C_VEL
LIN {X 0,Y 404.803,Z 536.805,A -85,B 0,C 180,E1 -10737.694,E2 -10737.694} C_VEL
LIN {X 0,Y 404.202,Z 534.132,A -85,B 0,C 180,E1 -10738.493,E2 -10738.493} C_VEL
LIN {X 0,Y 404.139,Z 534.142,A -85,B 0,C 180,E1 -10741.557,E2 -10741.557} C_VEL
LIN {X 0,Y 404.185,Z 534.138,A -85,B 0,C 180,E1 -10745.015,E2 -10745.015} C_VEL
LIN {X 0,Y 404.162,Z 534.143,A -85,B 0,C 180,E1 -10748.755,E2 -10748.755} C_VEL
LIN {X 0,Y 404.189,Z 534.134,A -85,B 0,C 180,E1 -10751.61,E2 -10751.61} C_VEL
LIN {X 0,Y 404.188,Z 534.14,A -85,B 0,C 180,E1 -10754.528,E2 -10754.528} C_VEL
LIN {X 0,Y 404.17,Z 534.136,A -85,B 0,C 180,E1 -10757.3,E2 -10757.3} C_VEL
LIN {X 0,Y 404.165,Z 534.132,A -85,B 0,C 180,E1 -10759.954,E2 -10759.954} C_VEL
LIN {X 0,Y 404.136,Z 534.142,A -85,B 0,C 180,E1 -10763.123,E2 -10763.123} C_VEL
LIN {X 0,Y 404.14,Z 534.141,A -85,B 0,C 180,E1 -10766.187,E2 -10766.187} C_VEL
LIN {X 0,Y 404.149,Z 534.135,A -85,B 0,C 180,E1 -10769.715,E2 -10769.715} C_VEL
LIN {X 0,Y 404.189,Z 534.132,A -85,B 0,C 180,E1 -10773.122,E2 -10773.122} C_VEL
LIN {X 0,Y 404.17,Z 534.138,A -85,B 0,C 180,E1 -10775.334,E2 -10775.334} C_VEL
LIN {X 0,Y 404.131,Z 534.142,A -85,B 0,C 180,E1 -10778.58,E2 -10778.58} C_VEL
LIN {X 0,Y 404.202,Z 534.13,A -85,B 0,C 180,E1 -10781.761,E2 -10781.761} C_VEL
LIN {X 0,Y 404.198,Z 534.137,A -85,B 0,C 180,E1 -10784.881,E2 -10784.881} C_VEL
LIN {X 0,Y 404.248,Z 534.122,A -85,B 0,C 180,E1 -10787.958,E2 -10787.958} C_VEL
LIN {X 0,Y 404.397,Z 534.107,A -85,B 0,C 180,E1 -10792.128,E2 -10792.128} C_VEL
LIN {X 0,Y 404.416,Z 534.105,A -85,B 0,C 180,E1 -10794.015,E2 -10794.015} C_VEL
LIN {X 0,Y 404.474,Z 534.093,A -85,B 0,C 180,E1 -10798.008,E2 -10798.008} C_VEL
LIN {X 0,Y 404.604,Z 534.083,A -85,B 0,C 180,E1 -10800,E2 -10800} C_VEL
LIN {X 0,Y 404.415,Z 534.102,A -85,B 0,C 180,E1 -10802.988,E2 -10802.988} C_VEL
LIN {X 0,Y 404.414,Z 534.107,A -85,B 0,C 180,E1 -10805.985,E2 -10805.985} C_VEL
LIN {X 0,Y 404.283,Z 534.123,A -85,B 0,C 180,E1 -10809.001,E2 -10809.001} C_VEL
LIN {X 0,Y 404.248,Z 534.128,A -85,B 0,C 180,E1 -10812.042,E2 -10812.042} C_VEL
LIN {X 0,Y 404.198,Z 534.135,A -85,B 0,C 180,E1 -10815.118,E2 -10815.118} C_VEL
LIN {X 0,Y 404.202,Z 534.133,A -85,B 0,C 180,E1 -10818.238,E2 -10818.238} C_VEL
LIN {X 0,Y 404.13,Z 534.141,A -85,B 0,C 180,E1 -10821.42,E2 -10821.42} C_VEL
LIN {X 0,Y 404.167,Z 534.143,A -85,B 0,C 180,E1 -10824.666,E2 -10824.666} C_VEL
LIN {X 0,Y 404.191,Z 534.131,A -85,B 0,C 180,E1 -10828,E2 -10828} C_VEL
LIN {X 0,Y 404.136,Z 534.141,A -85,B 0,C 180,E1 -10831.559,E2 -10831.559} C_VEL
LIN {X 0,Y 404.179,Z 534.138,A -85,B 0,C 180,E1 -10835.017,E2 -10835.017} C_VEL
LIN {X 0,Y 404.158,Z 534.143,A -85,B 0,C 180,E1 -10838.757,E2 -10838.757} C_VEL
LIN {X 0,Y 404.145,Z 534.141,A -85,B 0,C 180,E1 -10841.605,E2 -10841.605} C_VEL
LIN {X 0,Y 404.142,Z 534.146,A -85,B 0,C 180,E1 -10844.523,E2 -10844.523} C_VEL
LIN {X 0,Y 404.136,Z 534.143,A -85,B 0,C 180,E1 -10847.297,E2 -10847.297} C_VEL
LIN {X 0,Y 404.166,Z 534.139,A -85,B 0,C 180,E1 -10849.956,E2 -10849.956} C_VEL
LIN {X 0,Y 404.137,Z 534.144,A -85,B 0,C 180,E1 -10853.125,E2 -10853.125} C_VEL
LIN {X 0,Y 404.143,Z 534.143,A -85,B 0,C 180,E1 -10856.188,E2 -10856.188} C_VEL
LIN {X 0,Y 404.144,Z 534.144,A -85,B 0,C 180,E1 -10859.716,E2 -10859.716} C_VEL
LIN {X 0,Y 404.225,Z 534.267,A -85,B 0,C 180,E1 -10861.615,E2 -10861.615} C_VEL
LIN {X 0,Y 406.441,Z 544.391,A -85,B 0,C 180,E1 -10864.048,E2 -10864.048} C_VEL
LIN {X 0,Y 407.731,Z 552.338,A -85,B 0,C 180,E1 -10865.877,E2 -10865.877} C_VEL
LIN {X 0,Y 406.458,Z 567.243,A -85,B 0,C 180,E1 -10869.02,E2 -10869.02} C_VEL
LIN {X 0,Y 406.132,Z 571.988,A -85,B 0,C 180,E1 -10870.016,E2 -10870.016} C_VEL
LIN {X 0,Y 410.276,Z 595.766,A -85,B 0,C 180,E1 -10870.692,E2 -10870.692} C_VEL
LIN {X 0,Y 410.813,Z 600.881,A -85,B 0,C 180,E1 -10870.813,E2 -10870.813} C_VEL
LIN {X 0,Y 409.772,Z 680.673,A -85,B 0,C 180,E1 -10872.244,E2 -10872.244} C_VEL
LIN {X 0,Y 409.166,Z 693.758,A -85,B 0,C 180,E1 -10872.669,E2 -10872.669} C_VEL
LIN {X 0,Y 408.6,Z 704.684,A -85,B 0,C 180,E1 -10873.192,E2 -10873.192} C_VEL
LIN {X 0,Y 407.709,Z 717.196,A -85,B 0,C 180,E1 -10873.99,E2 -10873.99} C_VEL
LIN {X 0,Y 406.791,Z 728.904,A -85,B 0,C 180,E1 -10874.981,E2 -10874.981} C_VEL
LIN {X 0,Y 405.884,Z 739.422,A -85,B 0,C 180,E1 -10876.099,E2 -10876.099} C_VEL
LIN {X 0,Y 405.233,Z 748.029,A -85,B 0,C 180,E1 -10877.225,E2 -10877.225} C_VEL
LIN {X 0,Y 404.461,Z 755.971,A -85,B 0,C 180,E1 -10878.473,E2 -10878.473} C_VEL
LIN {X 0,Y 403.852,Z 763.758,A -85,B 0,C 180,E1 -10879.978,E2 -10879.978} C_VEL
LIN {X 0,Y 403.402,Z 770.001,A -85,B 0,C 180,E1 -10881.484,E2 -10881.484} C_VEL
LIN {X 0,Y 403.084,Z 774.976,A -85,B 0,C 180,E1 -10882.99,E2 -10882.99} C_VEL
LIN {X 0,Y 402.928,Z 778.827,A -85,B 0,C 180,E1 -10884.495,E2 -10884.495} C_VEL
LIN {X 0,Y 402.855,Z 781.659,A -85,B 0,C 180,E1 -10885.999,E2 -10885.999} C_VEL
LIN {X 0,Y 402.864,Z 783.95,A -85,B 0,C 180,E1 -10888.001,E2 -10888.001} C_VEL
LIN {X 0,Y 402.862,Z 784.509,A -85,B 0,C 180,E1 -10889,E2 -10889} C_VEL
LIN {X 0,Y 402.851,Z 784.638,A -85,B 0,C 180,E1 -10890,E2 -10890} C_VEL
LIN {X 0,Y 402.862,Z 784.368,A -85,B 0,C 180,E1 -10891,E2 -10891} C_VEL
LIN {X 0,Y 402.865,Z 783.713,A -85,B 0,C 180,E1 -10891.999,E2 -10891.999} C_VEL
LIN {X 0,Y 402.828,Z 782.666,A -85,B 0,C 180,E1 -10893,E2 -10893} C_VEL
LIN {X 0,Y 402.856,Z 781.173,A -85,B 0,C 180,E1 -10894.001,E2 -10894.001} C_VEL
LIN {X 0,Y 402.927,Z 778.137,A -85,B 0,C 180,E1 -10895.505,E2 -10895.505} C_VEL
LIN {X 0,Y 403.081,Z 774.04,A -85,B 0,C 180,E1 -10897.01,E2 -10897.01} C_VEL
LIN {X 0,Y 403.424,Z 767.753,A -85,B 0,C 180,E1 -10898.768,E2 -10898.768} C_VEL
LIN {X 0,Y 403.898,Z 760.905,A -85,B 0,C 180,E1 -10900.274,E2 -10900.274} C_VEL
LIN {X 0,Y 404.384,Z 753.916,A -85,B 0,C 180,E1 -10901.529,E2 -10901.529} C_VEL
LIN {X 0,Y 405.1,Z 745.502,A -85,B 0,C 180,E1 -10902.779,E2 -10902.779} C_VEL
LIN {X 0,Y 405.853,Z 735.119,A -85,B 0,C 180,E1 -10904.03,E2 -10904.03} C_VEL
LIN {X 0,Y 406.651,Z 723.4,A -85,B 0,C 180,E1 -10905.153,E2 -10905.153} C_VEL
LIN {X 0,Y 407.458,Z 711.762,A -85,B 0,C 180,E1 -10906.02,E2 -10906.02} C_VEL
LIN {X 0,Y 408.101,Z 699.648,A -85,B 0,C 180,E1 -10906.701,E2 -10906.701} C_VEL
LIN {X 0,Y 408.706,Z 686.485,A -85,B 0,C 180,E1 -10907.222,E2 -10907.222} C_VEL
LIN {X 0,Y 409.098,Z 673.832,A -85,B 0,C 180,E1 -10907.528,E2 -10907.528} C_VEL
LIN {X 0,Y 409.822,Z 598.784,A -85,B 0,C 180,E1 -10908.843,E2 -10908.843} C_VEL
LIN {X 0,Y 405.747,Z 572.156,A -85,B 0,C 180,E1 -10909.512,E2 -10909.512} C_VEL
LIN {X 0,Y 406.851,Z 555.925,A -85,B 0,C 180,E1 -10912.871,E2 -10912.871} C_VEL
LIN {X 0,Y 407.206,Z 550.133,A -85,B 0,C 180,E1 -10914.08,E2 -10914.08} C_VEL
LIN {X 0,Y 405.006,Z 538.021,A -85,B 0,C 180,E1 -10916.818,E2 -10916.818} C_VEL
LIN {X 0,Y 404.239,Z 534.134,A -85,B 0,C 180,E1 -10917.72,E2 -10917.72} C_VEL
LIN {X 0,Y 404.138,Z 534.146,A -85,B 0,C 180,E1 -10921.557,E2 -10921.557} C_VEL
LIN {X 0,Y 404.183,Z 534.136,A -85,B 0,C 180,E1 -10925.015,E2 -10925.015} C_VEL
LIN {X 0,Y 404.156,Z 534.138,A -85,B 0,C 180,E1 -10928.756,E2 -10928.756} C_VEL
LIN {X 0,Y 404.122,Z 534.147,A -85,B 0,C 180,E1 -10931.599,E2 -10931.599} C_VEL
LIN {X 0,Y 404.145,Z 534.139,A -85,B 0,C 180,E1 -10934.522,E2 -10934.522} C_VEL
LIN {X 0,Y 404.166,Z 534.141,A -85,B 0,C 180,E1 -10937.299,E2 -10937.299} C_VEL
LIN {X 0,Y 404.164,Z 534.138,A -85,B 0,C 180,E1 -10939.955,E2 -10939.955} C_VEL
LIN {X 0,Y 404.135,Z 534.143,A -85,B 0,C 180,E1 -10943.124,E2 -10943.124} C_VEL
LIN {X 0,Y 404.139,Z 534.14,A -85,B 0,C 180,E1 -10946.187,E2 -10946.187} C_VEL
LIN {X 0,Y 404.147,Z 534.143,A -85,B 0,C 180,E1 -10949.715,E2 -10949.715} C_VEL
LIN {X 0,Y 404.188,Z 534.137,A -85,B 0,C 180,E1 -10953.122,E2 -10953.122} C_VEL
LIN {X 0,Y 404.167,Z 534.142,A -85,B 0,C 180,E1 -10955.334,E2 -10955.334} C_VEL
LIN {X 0,Y 404.13,Z 534.141,A -85,B 0,C 180,E1 -10958.58,E2 -10958.58} C_VEL
LIN {X 0,Y 404.202,Z 534.135,A -85,B 0,C 180,E1 -10961.762,E2 -10961.762} C_VEL
LIN {X 0,Y 404.198,Z 534.134,A -85,B 0,C 180,E1 -10964.882,E2 -10964.882} C_VEL
LIN {X 0,Y 404.248,Z 534.128,A -85,B 0,C 180,E1 -10967.958,E2 -10967.958} C_VEL
LIN {X 0,Y 404.397,Z 534.108,A -85,B 0,C 180,E1 -10972.128,E2 -10972.128} C_VEL
LIN {X 0,Y 404.415,Z 534.106,A -85,B 0,C 180,E1 -10974.015,E2 -10974.015} C_VEL
LIN {X 0,Y 404.474,Z 534.099,A -85,B 0,C 180,E1 -10978.009,E2 -10978.009} C_VEL
LIN {X 0,Y 404.602,Z 534.083,A -85,B 0,C 180,E1 -10980,E2 -10980} C_VEL
LIN {X 0,Y 404.416,Z 534.107,A -85,B 0,C 180,E1 -10982.989,E2 -10982.989} C_VEL
LIN {X 0,Y 404.389,Z 534.109,A -85,B 0,C 180,E1 -10986.646,E2 -10986.646} C_VEL
LIN {X 0,Y 404.283,Z 534.124,A -85,B 0,C 180,E1 -10989.001,E2 -10989.001} C_VEL
LIN {X 0,Y 404.249,Z 534.127,A -85,B 0,C 180,E1 -10992.042,E2 -10992.042} C_VEL
LIN {X 0,Y 404.198,Z 534.136,A -85,B 0,C 180,E1 -10995.118,E2 -10995.118} C_VEL
LIN {X 0,Y 404.202,Z 534.132,A -85,B 0,C 180,E1 -10998.239,E2 -10998.239} C_VEL
LIN {X 0,Y 404.152,Z 534.145,A -85,B 0,C 180,E1 -11001.419,E2 -11001.419} C_VEL
LIN {X 0,Y 404.17,Z 534.136,A -85,B 0,C 180,E1 -11004.666,E2 -11004.666} C_VEL
LIN {X 0,Y 404.192,Z 534.134,A -85,B 0,C 180,E1 -11008,E2 -11008} C_VEL
LIN {X 0,Y 404.139,Z 534.145,A -85,B 0,C 180,E1 -11011.56,E2 -11011.56} C_VEL
LIN {X 0,Y 404.18,Z 534.137,A -85,B 0,C 180,E1 -11015.017,E2 -11015.017} C_VEL
LIN {X 0,Y 404.155,Z 534.138,A -85,B 0,C 180,E1 -11018.757,E2 -11018.757} C_VEL
LIN {X 0,Y 404.121,Z 534.147,A -85,B 0,C 180,E1 -11021.601,E2 -11021.601} C_VEL
LIN {X 0,Y 404.154,Z 534.138,A -85,B 0,C 180,E1 -11024.525,E2 -11024.525} C_VEL
LIN {X 0,Y 404.205,Z 534.138,A -85,B 0,C 180,E1 -11027.306,E2 -11027.306} C_VEL
LIN {X 0,Y 404.167,Z 534.137,A -85,B 0,C 180,E1 -11029.956,E2 -11029.956} C_VEL
LIN {X 0,Y 404.14,Z 534.143,A -85,B 0,C 180,E1 -11033.125,E2 -11033.125} C_VEL
LIN {X 0,Y 404.145,Z 534.139,A -85,B 0,C 180,E1 -11036.189,E2 -11036.189} C_VEL
LIN {X 0,Y 404.146,Z 534.142,A -85,B 0,C 180,E1 -11039.716,E2 -11039.716} C_VEL
LIN {X 0,Y 404.197,Z 534.136,A -85,B 0,C 180,E1 -11043.124,E2 -11043.124} C_VEL
LIN {X 0,Y 404.179,Z 534.141,A -85,B 0,C 180,E1 -11045.335,E2 -11045.335} C_VEL
LIN {X 0,Y 404.141,Z 534.145,A -85,B 0,C 180,E1 -11048.581,E2 -11048.581} C_VEL
LIN {X 0,Y 404.213,Z 534.16,A -85,B 0,C 180,E1 -11050.318,E2 -11050.318} C_VEL
LIN {X 0,Y 406.231,Z 545.041,A -85,B 0,C 180,E1 -11053.155,E2 -11053.155} C_VEL
LIN {X 0,Y 406,Z 550.85,A -85,B 0,C 180,E1 -11054.562,E2 -11054.562} C_VEL
LIN {X 0,Y 410.103,Z 572.048,A -85,B 0,C 180,E1 -11055.144,E2 -11055.144} C_VEL
LIN {X 0,Y 409.118,Z 657.33,A -85,B 0,C 180,E1 -11056.654,E2 -11056.654} C_VEL
LIN {X 0,Y 408.684,Z 670.648,A -85,B 0,C 180,E1 -11057.082,E2 -11057.082} C_VEL
LIN {X 0,Y 408.122,Z 683.359,A -85,B 0,C 180,E1 -11057.696,E2 -11057.696} C_VEL
LIN {X 0,Y 407.488,Z 694.661,A -85,B 0,C 180,E1 -11058.434,E2 -11058.434} C_VEL
LIN {X 0,Y 406.762,Z 706.275,A -85,B 0,C 180,E1 -11059.422,E2 -11059.422} C_VEL
LIN {X 0,Y 405.861,Z 716.721,A -85,B 0,C 180,E1 -11060.532,E2 -11060.532} C_VEL
LIN {X 0,Y 405.245,Z 725.865,A -85,B 0,C 180,E1 -11061.737,E2 -11061.737} C_VEL
LIN {X 0,Y 404.716,Z 733.826,A -85,B 0,C 180,E1 -11063.018,E2 -11063.018} C_VEL
LIN {X 0,Y 404.111,Z 741.365,A -85,B 0,C 180,E1 -11064.511,E2 -11064.511} C_VEL
LIN {X 0,Y 403.598,Z 747.435,A -85,B 0,C 180,E1 -11066.006,E2 -11066.006} C_VEL
LIN {X 0,Y 403.253,Z 752.253,A -85,B 0,C 180,E1 -11067.503,E2 -11067.503} C_VEL
LIN {X 0,Y 402.957,Z 755.969,A -85,B 0,C 180,E1 -11069.001,E2 -11069.001} C_VEL
LIN {X 0,Y 402.887,Z 757.886,A -85,B 0,C 180,E1 -11070,E2 -11070} C_VEL
LIN {X 0,Y 402.882,Z 759.538,A -85,B 0,C 180,E1 -11071.143,E2 -11071.143} C_VEL
LIN {X 0,Y 402.205,Z 760.44,A -85,B 0,C 180,E1 -11071.97,E2 -11071.97} C_VEL
LIN {X 0,Y 399.321,Z 761.364,A -85,B 0,C 180,E1 -11073.321,E2 -11073.321} C_VEL
LIN {X 0,Y 396.895,Z 761.583,A -85,B 0,C 180,E1 -11074.415,E2 -11074.415} C_VEL
LIN {X 0,Y 395.867,Z 761.415,A -85,B 0,C 180,E1 -11075.261,E2 -11075.261} C_VEL
LIN {X 0,Y 395.791,Z 761.25,A -85,B 0,C 180,E1 -11075.547,E2 -11075.547} C_VEL
LIN {X 0,Y 395.879,Z 760.012,A -85,B 0,C 180,E1 -11077.138,E2 -11077.138} C_VEL
LIN {X 0,Y 395.9,Z 758.688,A -85,B 0,C 180,E1 -11078.164,E2 -11078.164} C_VEL
LIN {X 0,Y 396.055,Z 755.875,A -85,B 0,C 180,E1 -11079.705,E2 -11079.705} C_VEL
LIN {X 0,Y 396.386,Z 752.029,A -85,B 0,C 180,E1 -11081.246,E2 -11081.246} C_VEL
LIN {X 0,Y 396.786,Z 746.791,A -85,B 0,C 180,E1 -11082.864,E2 -11082.864} C_VEL
LIN {X 0,Y 397.451,Z 739.534,A -85,B 0,C 180,E1 -11084.594,E2 -11084.594} C_VEL
LIN {X 0,Y 398.225,Z 731.363,A -85,B 0,C 180,E1 -11086.138,E2 -11086.138} C_VEL
LIN {X 0,Y 399.112,Z 722.989,A -85,B 0,C 180,E1 -11087.418,E2 -11087.418} C_VEL
LIN {X 0,Y 399.873,Z 713.81,A -85,B 0,C 180,E1 -11088.575,E2 -11088.575} C_VEL
LIN {X 0,Y 400.721,Z 703.787,A -85,B 0,C 180,E1 -11089.598,E2 -11089.598} C_VEL
LIN {X 0,Y 401.545,Z 692.86,A -85,B 0,C 180,E1 -11090.49,E2 -11090.49} C_VEL
LIN {X 0,Y 402.341,Z 680.77,A -85,B 0,C 180,E1 -11091.251,E2 -11091.251} C_VEL
LIN {X 0,Y 402.88,Z 669.261,A -85,B 0,C 180,E1 -11091.786,E2 -11091.786} C_VEL
LIN {X 0,Y 403.274,Z 657.4,A -85,B 0,C 180,E1 -11092.159,E2 -11092.159} C_VEL
LIN {X 0,Y 404.353,Z 572.934,A -85,B 0,C 180,E1 -11093.693,E2 -11093.693} C_VEL
LIN {X 0,Y 399.617,Z 551.161,A -85,B 0,C 180,E1 -11094.384,E2 -11094.384} C_VEL
LIN {X 0,Y 399.634,Z 547.781,A -85,B 0,C 180,E1 -11095.243,E2 -11095.243} C_VEL
LIN {X 0,Y 397.774,Z 537.86,A -85,B 0,C 180,E1 -11097.942,E2 -11097.942} C_VEL
LIN {X 0,Y 397.162,Z 535.01,A -85,B 0,C 180,E1 -11098.756,E2 -11098.756} C_VEL
LIN {X 0,Y 397.078,Z 535.023,A -85,B 0,C 180,E1 -11102.071,E2 -11102.071} C_VEL
LIN {X 0,Y 397.119,Z 535.017,A -85,B 0,C 180,E1 -11105.503,E2 -11105.503} C_VEL
LIN {X 0,Y 397.136,Z 535.019,A -85,B 0,C 180,E1 -11108.862,E2 -11108.862} C_VEL
LIN {X 0,Y 397.156,Z 535.013,A -85,B 0,C 180,E1 -11112.254,E2 -11112.254} C_VEL
LIN {X 0,Y 397.11,Z 535.018,A -85,B 0,C 180,E1 -11115.064,E2 -11115.064} C_VEL
LIN {X 0,Y 397.107,Z 535.016,A -85,B 0,C 180,E1 -11118.013,E2 -11118.013} C_VEL
LIN {X 0,Y 397.131,Z 535.016,A -85,B 0,C 180,E1 -11121.137,E2 -11121.137} C_VEL
LIN {X 0,Y 397.115,Z 535.02,A -85,B 0,C 180,E1 -11124.496,E2 -11124.496} C_VEL
LIN {X 0,Y 397.076,Z 535.021,A -85,B 0,C 180,E1 -11127.928,E2 -11127.928} C_VEL
LIN {X 0,Y 397.121,Z 535.015,A -85,B 0,C 180,E1 -11131.456,E2 -11131.456} C_VEL
LIN {X 0,Y 397.146,Z 535.012,A -85,B 0,C 180,E1 -11134.487,E2 -11134.487} C_VEL
LIN {X 0,Y 397.102,Z 535.014,A -85,B 0,C 180,E1 -11137.085,E2 -11137.085} C_VEL
LIN {X 0,Y 397.14,Z 535.016,A -85,B 0,C 180,E1 -11140.352,E2 -11140.352} C_VEL
LIN {X 0,Y 397.158,Z 535.009,A -85,B 0,C 180,E1 -11143.553,E2 -11143.553} C_VEL
LIN {X 0,Y 397.221,Z 535.001,A -85,B 0,C 180,E1 -11146.702,E2 -11146.702} C_VEL
LIN {X 0,Y 397.21,Z 535.004,A -85,B 0,C 180,E1 -11149.809,E2 -11149.809} C_VEL
LIN {X 0,Y 397.344,Z 534.986,A -85,B 0,C 180,E1 -11152.888,E2 -11152.888} C_VEL
LIN {X 0,Y 397.249,Z 535.002,A -85,B 0,C 180,E1 -11154.925,E2 -11154.925} C_VEL
LIN {X 0,Y 397.443,Z 534.969,A -85,B 0,C 180,E1 -11157.973,E2 -11157.973} C_VEL
LIN {X 0,Y 397.574,Z 534.959,A -85,B 0,C 180,E1 -11160,E2 -11160} C_VEL
LIN {X 0,Y 397.374,Z 534.979,A -85,B 0,C 180,E1 -11163.041,E2 -11163.041} C_VEL
LIN {X 0,Y 397.365,Z 534.986,A -85,B 0,C 180,E1 -11166.092,E2 -11166.092} C_VEL
LIN {X 0,Y 397.244,Z 534.998,A -85,B 0,C 180,E1 -11169.162,E2 -11169.162} C_VEL
LIN {X 0,Y 397.211,Z 535.007,A -85,B 0,C 180,E1 -11172.258,E2 -11172.258} C_VEL
LIN {X 0,Y 397.171,Z 535.009,A -85,B 0,C 180,E1 -11175.392,E2 -11175.392} C_VEL
LIN {X 0,Y 397.154,Z 535.01,A -85,B 0,C 180,E1 -11178.574,E2 -11178.574} C_VEL
LIN {X 0,Y 397.088,Z 535.019,A -85,B 0,C 180,E1 -11181.819,E2 -11181.819} C_VEL
LIN {X 0,Y 397.145,Z 535.011,A -85,B 0,C 180,E1 -11185.513,E2 -11185.513} C_VEL
LIN {X 0,Y 397.12,Z 535.017,A -85,B 0,C 180,E1 -11188.544,E2 -11188.544} C_VEL
LIN {X 0,Y 397.074,Z 535.022,A -85,B 0,C 180,E1 -11192.072,E2 -11192.072} C_VEL
LIN {X 0,Y 397.114,Z 535.016,A -85,B 0,C 180,E1 -11195.504,E2 -11195.504} C_VEL
LIN {X 0,Y 397.132,Z 535.017,A -85,B 0,C 180,E1 -11198.863,E2 -11198.863} C_VEL
LIN {X 0,Y 397.109,Z 535.021,A -85,B 0,C 180,E1 -11202.262,E2 -11202.262} C_VEL
LIN {X 0,Y 397.085,Z 535.022,A -85,B 0,C 180,E1 -11205.069,E2 -11205.069} C_VEL
LIN {X 0,Y 397.065,Z 535.025,A -85,B 0,C 180,E1 -11208.022,E2 -11208.022} C_VEL
LIN {X 0,Y 397.131,Z 535.016,A -85,B 0,C 180,E1 -11211.139,E2 -11211.139} C_VEL
LIN {X 0,Y 397.118,Z 535.018,A -85,B 0,C 180,E1 -11214.497,E2 -11214.497} C_VEL
LIN {X 0,Y 397.077,Z 535.025,A -85,B 0,C 180,E1 -11217.929,E2 -11217.929} C_VEL
LIN {X 0,Y 397.174,Z 535.165,A -85,B 0,C 180,E1 -11221.281,E2 -11221.281} C_VEL
LIN {X 0,Y 399.528,Z 545.877,A -85,B 0,C 180,E1 -11223.912,E2 -11223.912} C_VEL
LIN {X 0,Y 400.823,Z 553.713,A -85,B 0,C 180,E1 -11225.751,E2 -11225.751} C_VEL
LIN {X 0,Y 399.493,Z 568.636,A -85,B 0,C 180,E1 -11228.955,E2 -11228.955} C_VEL
LIN {X 0,Y 399.265,Z 571.844,A -85,B 0,C 180,E1 -11229.64,E2 -11229.64} C_VEL
LIN {X 0,Y 403.414,Z 595.257,A -85,B 0,C 180,E1 -11230.317,E2 -11230.317} C_VEL
LIN {X 0,Y 404.179,Z 600.674,A -85,B 0,C 180,E1 -11230.459,E2 -11230.459} C_VEL
LIN {X 0,Y 403.058,Z 680.253,A -85,B 0,C 180,E1 -11231.906,E2 -11231.906} C_VEL
LIN {X 0,Y 402.469,Z 693.406,A -85,B 0,C 180,E1 -11232.338,E2 -11232.338} C_VEL
LIN {X 0,Y 401.864,Z 703.807,A -85,B 0,C 180,E1 -11232.836,E2 -11232.836} C_VEL
LIN {X 0,Y 401.035,Z 715.594,A -85,B 0,C 180,E1 -11233.586,E2 -11233.586} C_VEL
LIN {X 0,Y 400.146,Z 726.327,A -85,B 0,C 180,E1 -11234.464,E2 -11234.464} C_VEL
LIN {X 0,Y 399.269,Z 736.39,A -85,B 0,C 180,E1 -11235.494,E2 -11235.494} C_VEL
LIN {X 0,Y 398.451,Z 746.218,A -85,B 0,C 180,E1 -11236.745,E2 -11236.745} C_VEL
LIN {X 0,Y 397.483,Z 755.912,A -85,B 0,C 180,E1 -11238.268,E2 -11238.268} C_VEL
LIN {X 0,Y 396.85,Z 763.662,A -85,B 0,C 180,E1 -11239.8,E2 -11239.8} C_VEL
LIN {X 0,Y 396.358,Z 769.884,A -85,B 0,C 180,E1 -11241.332,E2 -11241.332} C_VEL
LIN {X 0,Y 396.013,Z 774.839,A -85,B 0,C 180,E1 -11242.864,E2 -11242.864} C_VEL
LIN {X 0,Y 395.833,Z 778.232,A -85,B 0,C 180,E1 -11244.186,E2 -11244.186} C_VEL
LIN {X 0,Y 395.778,Z 781.489,A -85,B 0,C 180,E1 -11245.927,E2 -11245.927} C_VEL
LIN {X 0,Y 395.762,Z 783.764,A -85,B 0,C 180,E1 -11247.965,E2 -11247.965} C_VEL
LIN {X 0,Y 395.791,Z 784.314,A -85,B 0,C 180,E1 -11248.983,E2 -11248.983} C_VEL
LIN {X 0,Y 395.778,Z 784.43,A -85,B 0,C 180,E1 -11250,E2 -11250} C_VEL
LIN {X 0,Y 395.791,Z 784.153,A -85,B 0,C 180,E1 -11251.017,E2 -11251.017} C_VEL
LIN {X 0,Y 395.763,Z 783.489,A -85,B 0,C 180,E1 -11252.035,E2 -11252.035} C_VEL
LIN {X 0,Y 395.731,Z 782.432,A -85,B 0,C 180,E1 -11253.054,E2 -11253.054} C_VEL
LIN {X 0,Y 395.778,Z 780.926,A -85,B 0,C 180,E1 -11254.073,E2 -11254.073} C_VEL
LIN {X 0,Y 395.831,Z 777.36,A -85,B 0,C 180,E1 -11255.812,E2 -11255.812} C_VEL
LIN {X 0,Y 396.077,Z 772.13,A -85,B 0,C 180,E1 -11257.647,E2 -11257.647} C_VEL
LIN {X 0,Y 396.424,Z 766.431,A -85,B 0,C 180,E1 -11259.181,E2 -11259.181} C_VEL
LIN {X 0,Y 396.908,Z 759.275,A -85,B 0,C 180,E1 -11260.715,E2 -11260.715} C_VEL
LIN {X 0,Y 397.685,Z 750.363,A -85,B 0,C 180,E1 -11262.243,E2 -11262.243} C_VEL
LIN {X 0,Y 398.387,Z 741.374,A -85,B 0,C 180,E1 -11263.496,E2 -11263.496} C_VEL
LIN {X 0,Y 399.192,Z 731.219,A -85,B 0,C 180,E1 -11264.646,E2 -11264.646} C_VEL
LIN {X 0,Y 399.966,Z 719.816,A -85,B 0,C 180,E1 -11265.674,E2 -11265.674} C_VEL
LIN {X 0,Y 400.862,Z 707.161,A -85,B 0,C 180,E1 -11266.552,E2 -11266.552} C_VEL
LIN {X 0,Y 401.514,Z 694.814,A -85,B 0,C 180,E1 -11267.18,E2 -11267.18} C_VEL
LIN {X 0,Y 402.096,Z 681.078,A -85,B 0,C 180,E1 -11267.646,E2 -11267.646} C_VEL
LIN {X 0,Y 402.74,Z 634.861,A -85,B 0,C 180,E1 -11268.496,E2 -11268.496} C_VEL
LIN {X 0,Y 402.933,Z 598.518,A -85,B 0,C 180,E1 -11269.152,E2 -11269.152} C_VEL
LIN {X 0,Y 398.794,Z 571.825,A -85,B 0,C 180,E1 -11269.864,E2 -11269.864} C_VEL
LIN {X 0,Y 400.027,Z 555.599,A -85,B 0,C 180,E1 -11273.284,E2 -11273.284} C_VEL
LIN {X 0,Y 400.28,Z 551.872,A -85,B 0,C 180,E1 -11274.076,E2 -11274.076} C_VEL
LIN {X 0,Y 398.49,Z 541.539,A -85,B 0,C 180,E1 -11276.443,E2 -11276.443} C_VEL
LIN {X 0,Y 397.172,Z 535.014,A -85,B 0,C 180,E1 -11278.004,E2 -11278.004} C_VEL
LIN {X 0,Y 397.078,Z 535.025,A -85,B 0,C 180,E1 -11280.882,E2 -11280.882} C_VEL
LIN {X 0,Y 397.124,Z 535.013,A -85,B 0,C 180,E1 -11284.492,E2 -11284.492} C_VEL
LIN {X 0,Y 397.104,Z 535.016,A -85,B 0,C 180,E1 -11288.274,E2 -11288.274} C_VEL
LIN {X 0,Y 397.087,Z 535.019,A -85,B 0,C 180,E1 -11290.908,E2 -11290.908} C_VEL
LIN {X 0,Y 397.1,Z 535.021,A -85,B 0,C 180,E1 -11293.647,E2 -11293.647} C_VEL
LIN {X 0,Y 397.1,Z 535.016,A -85,B 0,C 180,E1 -11296.52,E2 -11296.52} C_VEL
LIN {X 0,Y 397.115,Z 535.021,A -85,B 0,C 180,E1 -11299.551,E2 -11299.551} C_VEL
LIN {X 0,Y 397.093,Z 535.018,A -85,B 0,C 180,E1 -11302.789,E2 -11302.789} C_VEL
LIN {X 0,Y 397.112,Z 535.015,A -85,B 0,C 180,E1 -11306.281,E2 -11306.281} C_VEL
LIN {X 0,Y 397.107,Z 535.016,A -85,B 0,C 180,E1 -11310.133,E2 -11310.133} C_VEL
LIN {X 0,Y 397.188,Z 535.006,A -85,B 0,C 180,E1 -11312.609,E2 -11312.609} C_VEL
LIN {X 0,Y 397.121,Z 535.015,A -85,B 0,C 180,E1 -11315.981,E2 -11315.981} C_VEL
LIN {X 0,Y 397.131,Z 535.017,A -85,B 0,C 180,E1 -11319.704,E2 -11319.704} C_VEL
LIN {X 0,Y 397.174,Z 535.008,A -85,B 0,C 180,E1 -11322.845,E2 -11322.845} C_VEL
LIN {X 0,Y 397.22,Z 535.002,A -85,B 0,C 180,E1 -11326.702,E2 -11326.702} C_VEL
LIN {X 0,Y 397.21,Z 535.006,A -85,B 0,C 180,E1 -11329.809,E2 -11329.809} C_VEL
LIN {X 0,Y 397.347,Z 534.987,A -85,B 0,C 180,E1 -11332.888,E2 -11332.888} C_VEL
LIN {X 0,Y 397.248,Z 535,A -85,B 0,C 180,E1 -11334.925,E2 -11334.925} C_VEL
LIN {X 0,Y 397.443,Z 534.975,A -85,B 0,C 180,E1 -11337.973,E2 -11337.973} C_VEL
LIN {X 0,Y 397.571,Z 534.959,A -85,B 0,C 180,E1 -11340,E2 -11340} C_VEL
LIN {X 0,Y 397.374,Z 534.985,A -85,B 0,C 180,E1 -11343.042,E2 -11343.042} C_VEL
LIN {X 0,Y 397.34,Z 534.987,A -85,B 0,C 180,E1 -11346.644,E2 -11346.644} C_VEL
LIN {X 0,Y 397.245,Z 535.002,A -85,B 0,C 180,E1 -11349.162,E2 -11349.162} C_VEL
LIN {X 0,Y 397.211,Z 535.003,A -85,B 0,C 180,E1 -11352.259,E2 -11352.259} C_VEL
LIN {X 0,Y 397.171,Z 535.015,A -85,B 0,C 180,E1 -11355.393,E2 -11355.393} C_VEL
LIN {X 0,Y 397.154,Z 535.01,A -85,B 0,C 180,E1 -11358.574,E2 -11358.574} C_VEL
LIN {X 0,Y 397.101,Z 535.019,A -85,B 0,C 180,E1 -11361.818,E2 -11361.818} C_VEL
LIN {X 0,Y 397.146,Z 535.017,A -85,B 0,C 180,E1 -11365.513,E2 -11365.513} C_VEL
LIN {X 0,Y 397.12,Z 535.014,A -85,B 0,C 180,E1 -11368.544,E2 -11368.544} C_VEL
LIN {X 0,Y 397.076,Z 535.02,A -85,B 0,C 180,E1 -11372.072,E2 -11372.072} C_VEL
LIN {X 0,Y 397.115,Z 535.021,A -85,B 0,C 180,E1 -11375.504,E2 -11375.504} C_VEL
LIN {X 0,Y 397.129,Z 535.014,A -85,B 0,C 180,E1 -11378.863,E2 -11378.863} C_VEL
LIN {X 0,Y 397.068,Z 535.021,A -85,B 0,C 180,E1 -11382.268,E2 -11382.268} C_VEL
LIN {X 0,Y 397.115,Z 535.018,A -85,B 0,C 180,E1 -11385.065,E2 -11385.065} C_VEL
LIN {X 0,Y 397.154,Z 535.011,A -85,B 0,C 180,E1 -11388.008,E2 -11388.008} C_VEL
LIN {X 0,Y 397.109,Z 535.019,A -85,B 0,C 180,E1 -11391.727,E2 -11391.727} C_VEL
LIN {X 0,Y 397.125,Z 535.019,A -85,B 0,C 180,E1 -11395.508,E2 -11395.508} C_VEL
LIN {X 0,Y 397.079,Z 535.023,A -85,B 0,C 180,E1 -11399.118,E2 -11399.118} C_VEL
LIN {X 0,Y 397.195,Z 535.005,A -85,B 0,C 180,E1 -11402.611,E2 -11402.611} C_VEL
LIN {X 0,Y 397.135,Z 535.013,A -85,B 0,C 180,E1 -11405.983,E2 -11405.983} C_VEL
LIN {X 0,Y 397.163,Z 535.018,A -85,B 0,C 180,E1 -11410.061,E2 -11410.061} C_VEL
LIN {X 0,Y 399.15,Z 545.44,A -85,B 0,C 180,E1 -11412.847,E2 -11412.847} C_VEL
LIN {X 0,Y 399.129,Z 550.523,A -85,B 0,C 180,E1 -11414.109,E2 -11414.109} C_VEL
LIN {X 0,Y 399.101,Z 551.087,A -85,B 0,C 180,E1 -11414.247,E2 -11414.247} C_VEL
LIN {X 0,Y 403.324,Z 572.698,A -85,B 0,C 180,E1 -11414.849,E2 -11414.849} C_VEL
LIN {X 0,Y 402.311,Z 658.082,A -85,B 0,C 180,E1 -11416.392,E2 -11416.392} C_VEL
LIN {X 0,Y 401.843,Z 671.212,A -85,B 0,C 180,E1 -11416.826,E2 -11416.826} C_VEL
LIN {X 0,Y 401.309,Z 683.267,A -85,B 0,C 180,E1 -11417.42,E2 -11417.42} C_VEL
LIN {X 0,Y 400.585,Z 695.456,A -85,B 0,C 180,E1 -11418.232,E2 -11418.232} C_VEL
LIN {X 0,Y 399.835,Z 706.953,A -85,B 0,C 180,E1 -11419.237,E2 -11419.237} C_VEL
LIN {X 0,Y 398.91,Z 717.318,A -85,B 0,C 180,E1 -11420.365,E2 -11420.365} C_VEL
LIN {X 0,Y 398.367,Z 724.846,A -85,B 0,C 180,E1 -11421.369,E2 -11421.369} C_VEL
LIN {X 0,Y 397.718,Z 732.852,A -85,B 0,C 180,E1 -11422.64,E2 -11422.64} C_VEL
LIN {X 0,Y 397.124,Z 740.666,A -85,B 0,C 180,E1 -11424.16,E2 -11424.16} C_VEL
LIN {X 0,Y 396.71,Z 745.959,A -85,B 0,C 180,E1 -11425.428,E2 -11425.428} C_VEL
LIN {X 0,Y 396.236,Z 751.147,A -85,B 0,C 180,E1 -11426.95,E2 -11426.95} C_VEL
LIN {X 0,Y 396.015,Z 755.177,A -85,B 0,C 180,E1 -11428.475,E2 -11428.475} C_VEL
LIN {X 0,Y 395.812,Z 758.173,A -85,B 0,C 180,E1 -11430,E2 -11430} C_VEL
LIN {X 0,Y 395.807,Z 759.764,A -85,B 0,C 180,E1 -11431.132,E2 -11431.132} C_VEL
LIN {X 0,Y 395.751,Z 761.338,A -85,B 0,C 180,E1 -11433.054,E2 -11433.054} C_VEL
LIN {X 0,Y 395.746,Z 761.612,A -85,B 0,C 180,E1 -11434.073,E2 -11434.073} C_VEL
LIN {X 0,Y 395.791,Z 761.25,A -85,B 0,C 180,E1 -11435.547,E2 -11435.547} C_VEL
LIN {X 0,Y 395.147,Z 760.769,A -85,B 0,C 180,E1 -11436.395,E2 -11436.395} C_VEL
LIN {X 0,Y 392.336,Z 759.456,A -85,B 0,C 180,E1 -11437.768,E2 -11437.768} C_VEL
LIN {X 0,Y 389.994,Z 757.93,A -85,B 0,C 180,E1 -11438.863,E2 -11438.863} C_VEL
LIN {X 0,Y 389.046,Z 756.383,A -85,B 0,C 180,E1 -11439.695,E2 -11439.695} C_VEL
LIN {X 0,Y 389,Z 755.779,A -85,B 0,C 180,E1 -11439.973,E2 -11439.973} C_VEL
LIN {X 0,Y 389.358,Z 752.103,A -85,B 0,C 180,E1 -11441.452,E2 -11441.452} C_VEL
LIN {X 0,Y 389.822,Z 746.432,A -85,B 0,C 180,E1 -11443.205,E2 -11443.205} C_VEL
LIN {X 0,Y 390.523,Z 739.513,A -85,B 0,C 180,E1 -11444.859,E2 -11444.859} C_VEL
LIN {X 0,Y 391.352,Z 731.295,A -85,B 0,C 180,E1 -11446.43,E2 -11446.43} C_VEL
LIN {X 0,Y 392.263,Z 722.863,A -85,B 0,C 180,E1 -11447.733,E2 -11447.733} C_VEL
LIN {X 0,Y 393.165,Z 712.41,A -85,B 0,C 180,E1 -11449.039,E2 -11449.039} C_VEL
LIN {X 0,Y 394.207,Z 700.6,A -85,B 0,C 180,E1 -11450.207,E2 -11450.207} C_VEL
LIN {X 0,Y 395.139,Z 688.72,A -85,B 0,C 180,E1 -11451.11,E2 -11451.11} C_VEL
LIN {X 0,Y 395.863,Z 676.303,A -85,B 0,C 180,E1 -11451.821,E2 -11451.821} C_VEL
LIN {X 0,Y 396.423,Z 663.76,A -85,B 0,C 180,E1 -11452.327,E2 -11452.327} C_VEL
LIN {X 0,Y 396.746,Z 650.286,A -85,B 0,C 180,E1 -11452.653,E2 -11452.653} C_VEL
LIN {X 0,Y 397.763,Z 573.887,A -85,B 0,C 180,E1 -11454.046,E2 -11454.046} C_VEL
LIN {X 0,Y 392.763,Z 551.352,A -85,B 0,C 180,E1 -11454.788,E2 -11454.788} C_VEL
LIN {X 0,Y 392.368,Z 547.223,A -85,B 0,C 180,E1 -11455.888,E2 -11455.888} C_VEL
LIN {X 0,Y 390.309,Z 536.793,A -85,B 0,C 180,E1 -11458.807,E2 -11458.807} C_VEL
LIN {X 0,Y 390.096,Z 535.894,A -85,B 0,C 180,E1 -11459.106,E2 -11459.106} C_VEL
LIN {X 0,Y 390.043,Z 535.901,A -85,B 0,C 180,E1 -11462.721,E2 -11462.721} C_VEL
LIN {X 0,Y 390.057,Z 535.897,A -85,B 0,C 180,E1 -11465.825,E2 -11465.825} C_VEL
LIN {X 0,Y 390.073,Z 535.897,A -85,B 0,C 180,E1 -11469.218,E2 -11469.218} C_VEL
LIN {X 0,Y 390.118,Z 535.891,A -85,B 0,C 180,E1 -11472.386,E2 -11472.386} C_VEL
LIN {X 0,Y 390.061,Z 535.895,A -85,B 0,C 180,E1 -11475.356,E2 -11475.356} C_VEL
LIN {X 0,Y 390.065,Z 535.892,A -85,B 0,C 180,E1 -11478.191,E2 -11478.191} C_VEL
LIN {X 0,Y 390.09,Z 535.896,A -85,B 0,C 180,E1 -11480.907,E2 -11480.907} C_VEL
LIN {X 0,Y 390.081,Z 535.896,A -85,B 0,C 180,E1 -11484.792,E2 -11484.792} C_VEL
LIN {X 0,Y 390.023,Z 535.904,A -85,B 0,C 180,E1 -11488.495,E2 -11488.495} C_VEL
LIN {X 0,Y 390.111,Z 535.89,A -85,B 0,C 180,E1 -11492.069,E2 -11492.069} C_VEL
LIN {X 0,Y 390.073,Z 535.893,A -85,B 0,C 180,E1 -11495.519,E2 -11495.519} C_VEL
LIN {X 0,Y 390.048,Z 535.9,A -85,B 0,C 180,E1 -11498.877,E2 -11498.877} C_VEL
LIN {X 0,Y 390.12,Z 535.885,A -85,B 0,C 180,E1 -11502.166,E2 -11502.166} C_VEL
LIN {X 0,Y 390.136,Z 535.885,A -85,B 0,C 180,E1 -11505.392,E2 -11505.392} C_VEL
LIN {X 0,Y 390.141,Z 535.885,A -85,B 0,C 180,E1 -11508.571,E2 -11508.571} C_VEL
LIN {X 0,Y 390.299,Z 535.862,A -85,B 0,C 180,E1 -11512.031,E2 -11512.031} C_VEL
LIN {X 0,Y 390.22,Z 535.879,A -85,B 0,C 180,E1 -11514.833,E2 -11514.833} C_VEL
LIN {X 0,Y 390.412,Z 535.844,A -85,B 0,C 180,E1 -11517.937,E2 -11517.937} C_VEL
LIN {X 0,Y 390.543,Z 535.834,A -85,B 0,C 180,E1 -11520,E2 -11520} C_VEL
LIN {X 0,Y 390.308,Z 535.859,A -85,B 0,C 180,E1 -11523.096,E2 -11523.096} C_VEL
LIN {X 0,Y 390.319,Z 535.865,A -85,B 0,C 180,E1 -11526.202,E2 -11526.202} C_VEL
LIN {X 0,Y 390.197,Z 535.875,A -85,B 0,C 180,E1 -11529.329,E2 -11529.329} C_VEL
LIN {X 0,Y 390.186,Z 535.872,A -85,B 0,C 180,E1 -11533.439,E2 -11533.439} C_VEL
LIN {X 0,Y 390.14,Z 535.882,A -85,B 0,C 180,E1 -11537.308,E2 -11537.308} C_VEL
LIN {X 0,Y 390.079,Z 535.896,A -85,B 0,C 180,E1 -11540.47,E2 -11540.47} C_VEL
LIN {X 0,Y 390.07,Z 535.896,A -85,B 0,C 180,E1 -11544.481,E2 -11544.481} C_VEL
LIN {X 0,Y 390.109,Z 535.885,A -85,B 0,C 180,E1 -11548.026,E2 -11548.026} C_VEL
LIN {X 0,Y 390.021,Z 535.899,A -85,B 0,C 180,E1 -11551.505,E2 -11551.505} C_VEL
LIN {X 0,Y 390.08,Z 535.893,A -85,B 0,C 180,E1 -11555.207,E2 -11555.207} C_VEL
LIN {X 0,Y 390.09,Z 535.893,A -85,B 0,C 180,E1 -11559.092,E2 -11559.092} C_VEL
LIN {X 0,Y 390.076,Z 535.899,A -85,B 0,C 180,E1 -11562.381,E2 -11562.381} C_VEL
LIN {X 0,Y 390.053,Z 535.899,A -85,B 0,C 180,E1 -11566.114,E2 -11566.114} C_VEL
LIN {X 0,Y 390.054,Z 535.896,A -85,B 0,C 180,E1 -11569.561,E2 -11569.561} C_VEL
LIN {X 0,Y 390.043,Z 535.899,A -85,B 0,C 180,E1 -11572.449,E2 -11572.449} C_VEL
LIN {X 0,Y 390.066,Z 535.896,A -85,B 0,C 180,E1 -11576.046,E2 -11576.046} C_VEL
LIN {X 0,Y 390.045,Z 535.901,A -85,B 0,C 180,E1 -11579.87,E2 -11579.87} C_VEL
LIN {X 0,Y 390.106,Z 535.907,A -85,B 0,C 180,E1 -11580.895,E2 -11580.895} C_VEL
LIN {X 0,Y 392.417,Z 546.556,A -85,B 0,C 180,E1 -11583.57,E2 -11583.57} C_VEL
LIN {X 0,Y 393.882,Z 554.583,A -85,B 0,C 180,E1 -11585.504,E2 -11585.504} C_VEL
LIN {X 0,Y 392.745,Z 567.46,A -85,B 0,C 180,E1 -11588.329,E2 -11588.329} C_VEL
LIN {X 0,Y 392.397,Z 571.604,A -85,B 0,C 180,E1 -11589.232,E2 -11589.232} C_VEL
LIN {X 0,Y 396.815,Z 596.287,A -85,B 0,C 180,E1 -11589.971,E2 -11589.971} C_VEL
LIN {X 0,Y 397.529,Z 601.885,A -85,B 0,C 180,E1 -11590.117,E2 -11590.117} C_VEL
LIN {X 0,Y 396.36,Z 679.854,A -85,B 0,C 180,E1 -11591.555,E2 -11591.555} C_VEL
LIN {X 0,Y 395.782,Z 693.067,A -85,B 0,C 180,E1 -11591.996,E2 -11591.996} C_VEL
LIN {X 0,Y 395.093,Z 704.067,A -85,B 0,C 180,E1 -11592.532,E2 -11592.532} C_VEL
LIN {X 0,Y 394.237,Z 715.751,A -85,B 0,C 180,E1 -11593.295,E2 -11593.295} C_VEL
LIN {X 0,Y 393.296,Z 726.41,A -85,B 0,C 180,E1 -11594.187,E2 -11594.187} C_VEL
LIN {X 0,Y 392.32,Z 737.117,A -85,B 0,C 180,E1 -11595.32,E2 -11595.32} C_VEL
LIN {X 0,Y 391.523,Z 746.193,A -85,B 0,C 180,E1 -11596.506,E2 -11596.506} C_VEL
LIN {X 0,Y 390.521,Z 755.856,A -85,B 0,C 180,E1 -11598.056,E2 -11598.056} C_VEL
LIN {X 0,Y 389.837,Z 763.568,A -85,B 0,C 180,E1 -11599.614,E2 -11599.614} C_VEL
LIN {X 0,Y 389.329,Z 769.769,A -85,B 0,C 180,E1 -11601.174,E2 -11601.174} C_VEL
LIN {X 0,Y 388.943,Z 774.704,A -85,B 0,C 180,E1 -11602.734,E2 -11602.734} C_VEL
LIN {X 0,Y 388.733,Z 778.403,A -85,B 0,C 180,E1 -11604.237,E2 -11604.237} C_VEL
LIN {X 0,Y 388.703,Z 781.32,A -85,B 0,C 180,E1 -11605.853,E2 -11605.853} C_VEL
LIN {X 0,Y 388.66,Z 783.579,A -85,B 0,C 180,E1 -11607.927,E2 -11607.927} C_VEL
LIN {X 0,Y 388.703,Z 784.117,A -85,B 0,C 180,E1 -11608.964,E2 -11608.964} C_VEL
LIN {X 0,Y 388.707,Z 784.222,A -85,B 0,C 180,E1 -11610,E2 -11610} C_VEL
LIN {X 0,Y 388.703,Z 783.937,A -85,B 0,C 180,E1 -11611.036,E2 -11611.036} C_VEL
LIN {X 0,Y 388.662,Z 783.264,A -85,B 0,C 180,E1 -11612.073,E2 -11612.073} C_VEL
LIN {X 0,Y 388.638,Z 782.197,A -85,B 0,C 180,E1 -11613.11,E2 -11613.11} C_VEL
LIN {X 0,Y 388.703,Z 780.677,A -85,B 0,C 180,E1 -11614.147,E2 -11614.147} C_VEL
LIN {X 0,Y 388.731,Z 777.474,A -85,B 0,C 180,E1 -11615.761,E2 -11615.761} C_VEL
LIN {X 0,Y 388.938,Z 773.471,A -85,B 0,C 180,E1 -11617.267,E2 -11617.267} C_VEL
LIN {X 0,Y 389.32,Z 767.143,A -85,B 0,C 180,E1 -11619.088,E2 -11619.088} C_VEL
LIN {X 0,Y 389.814,Z 760.248,A -85,B 0,C 180,E1 -11620.649,E2 -11620.649} C_VEL
LIN {X 0,Y 390.548,Z 751.63,A -85,B 0,C 180,E1 -11622.207,E2 -11622.207} C_VEL
LIN {X 0,Y 391.29,Z 742.775,A -85,B 0,C 180,E1 -11623.503,E2 -11623.503} C_VEL
LIN {X 0,Y 392.202,Z 731.873,A -85,B 0,C 180,E1 -11624.794,E2 -11624.794} C_VEL
LIN {X 0,Y 393.009,Z 720.879,A -85,B 0,C 180,E1 -11625.825,E2 -11625.825} C_VEL
LIN {X 0,Y 393.934,Z 708.551,A -85,B 0,C 180,E1 -11626.719,E2 -11626.719} C_VEL
LIN {X 0,Y 394.566,Z 696.879,A -85,B 0,C 180,E1 -11627.358,E2 -11627.358} C_VEL
LIN {X 0,Y 395.172,Z 684.512,A -85,B 0,C 180,E1 -11627.832,E2 -11627.832} C_VEL
LIN {X 0,Y 395.471,Z 670.498,A -85,B 0,C 180,E1 -11628.152,E2 -11628.152} C_VEL
LIN {X 0,Y 396.304,Z 600.489,A -85,B 0,C 180,E1 -11629.417,E2 -11629.417} C_VEL
LIN {X 0,Y 391.91,Z 571.646,A -85,B 0,C 180,E1 -11630.194,E2 -11630.194} C_VEL
LIN {X 0,Y 393.314,Z 554.005,A -85,B 0,C 180,E1 -11633.985,E2 -11633.985} C_VEL
LIN {X 0,Y 392.705,Z 548.891,A -85,B 0,C 180,E1 -11635.152,E2 -11635.152} C_VEL
LIN {X 0,Y 390.121,Z 535.891,A -85,B 0,C 180,E1 -11638.26,E2 -11638.26} C_VEL
LIN {X 0,Y 390.03,Z 535.898,A -85,B 0,C 180,E1 -11642.124,E2 -11642.124} C_VEL
LIN {X 0,Y 390.083,Z 535.894,A -85,B 0,C 180,E1 -11645.206,E2 -11645.206} C_VEL
LIN {X 0,Y 390.09,Z 535.893,A -85,B 0,C 180,E1 -11649.091,E2 -11649.091} C_VEL
LIN {X 0,Y 390.041,Z 535.896,A -85,B 0,C 180,E1 -11652.374,E2 -11652.374} C_VEL
LIN {X 0,Y 390.041,Z 535.901,A -85,B 0,C 180,E1 -11655.354,E2 -11655.354} C_VEL
LIN {X 0,Y 390.063,Z 535.893,A -85,B 0,C 180,E1 -11658.191,E2 -11658.191} C_VEL
LIN {X 0,Y 390.09,Z 535.891,A -85,B 0,C 180,E1 -11660.908,E2 -11660.908} C_VEL
LIN {X 0,Y 390.08,Z 535.892,A -85,B 0,C 180,E1 -11664.793,E2 -11664.793} C_VEL
LIN {X 0,Y 390.021,Z 535.898,A -85,B 0,C 180,E1 -11668.495,E2 -11668.495} C_VEL
LIN {X 0,Y 390.11,Z 535.888,A -85,B 0,C 180,E1 -11672.069,E2 -11672.069} C_VEL
LIN {X 0,Y 390.071,Z 535.898,A -85,B 0,C 180,E1 -11675.519,E2 -11675.519} C_VEL
LIN {X 0,Y 390.079,Z 535.897,A -85,B 0,C 180,E1 -11679.53,E2 -11679.53} C_VEL
LIN {X 0,Y 390.13,Z 535.889,A -85,B 0,C 180,E1 -11683.248,E2 -11683.248} C_VEL
LIN {X 0,Y 390.186,Z 535.878,A -85,B 0,C 180,E1 -11686.561,E2 -11686.561} C_VEL
LIN {X 0,Y 390.197,Z 535.877,A -85,B 0,C 180,E1 -11690.671,E2 -11690.671} C_VEL
LIN {X 0,Y 390.32,Z 535.864,A -85,B 0,C 180,E1 -11693.798,E2 -11693.798} C_VEL
LIN {X 0,Y 390.412,Z 535.851,A -85,B 0,C 180,E1 -11697.937,E2 -11697.937} C_VEL
LIN {X 0,Y 390.541,Z 535.835,A -85,B 0,C 180,E1 -11700,E2 -11700} C_VEL
LIN {X 0,Y 390.309,Z 535.866,A -85,B 0,C 180,E1 -11703.097,E2 -11703.097} C_VEL
LIN {X 0,Y 390.295,Z 535.864,A -85,B 0,C 180,E1 -11706.639,E2 -11706.639} C_VEL
LIN {X 0,Y 390.197,Z 535.882,A -85,B 0,C 180,E1 -11709.329,E2 -11709.329} C_VEL
LIN {X 0,Y 390.163,Z 535.881,A -85,B 0,C 180,E1 -11712.484,E2 -11712.484} C_VEL
LIN {X 0,Y 390.131,Z 535.889,A -85,B 0,C 180,E1 -11715.677,E2 -11715.677} C_VEL
LIN {X 0,Y 390.098,Z 535.891,A -85,B 0,C 180,E1 -11718.923,E2 -11718.923} C_VEL
LIN {X 0,Y 390.04,Z 535.896,A -85,B 0,C 180,E1 -11722.234,E2 -11722.234} C_VEL
LIN {X 0,Y 390.113,Z 535.89,A -85,B 0,C 180,E1 -11725.744,E2 -11725.744} C_VEL
LIN {X 0,Y 390.06,Z 535.897,A -85,B 0,C 180,E1 -11729.11,E2 -11729.11} C_VEL
LIN {X 0,Y 390.039,Z 535.897,A -85,B 0,C 180,E1 -11732.722,E2 -11732.722} C_VEL
LIN {X 0,Y 390.052,Z 535.897,A -85,B 0,C 180,E1 -11735.826,E2 -11735.826} C_VEL
LIN {X 0,Y 390.068,Z 535.897,A -85,B 0,C 180,E1 -11739.22,E2 -11739.22} C_VEL
LIN {X 0,Y 390.041,Z 535.896,A -85,B 0,C 180,E1 -11742.375,E2 -11742.375} C_VEL
LIN {X 0,Y 390.1,Z 535.889,A -85,B 0,C 180,E1 -11746.108,E2 -11746.108} C_VEL
LIN {X 0,Y 390.081,Z 535.895,A -85,B 0,C 180,E1 -11749.175,E2 -11749.175} C_VEL
LIN {X 0,Y 390.046,Z 535.895,A -85,B 0,C 180,E1 -11752.449,E2 -11752.449} C_VEL
LIN {X 0,Y 390.067,Z 535.893,A -85,B 0,C 180,E1 -11756.046,E2 -11756.046} C_VEL
LIN {X 0,Y 390.047,Z 535.897,A -85,B 0,C 180,E1 -11759.87,E2 -11759.87} C_VEL
LIN {X 0,Y 390.115,Z 535.892,A -85,B 0,C 180,E1 -11763.233,E2 -11763.233} C_VEL
LIN {X 0,Y 390.108,Z 535.888,A -85,B 0,C 180,E1 -11766.751,E2 -11766.751} C_VEL
LIN {X 0,Y 390.138,Z 536.008,A -85,B 0,C 180,E1 -11769.863,E2 -11769.863} C_VEL
LIN {X 0,Y 392.2,Z 546.885,A -85,B 0,C 180,E1 -11772.803,E2 -11772.803} C_VEL
LIN {X 0,Y 392.184,Z 551.327,A -85,B 0,C 180,E1 -11773.917,E2 -11773.917} C_VEL
LIN {X 0,Y 396.614,Z 574.23,A -85,B 0,C 180,E1 -11774.563,E2 -11774.563} C_VEL
LIN {X 0,Y 395.509,Z 658.801,A -85,B 0,C 180,E1 -11776.12,E2 -11776.12} C_VEL
LIN {X 0,Y 395.026,Z 671.761,A -85,B 0,C 180,E1 -11776.562,E2 -11776.562} C_VEL
LIN {X 0,Y 394.425,Z 684.29,A -85,B 0,C 180,E1 -11777.196,E2 -11777.196} C_VEL
LIN {X 0,Y 393.691,Z 696.233,A -85,B 0,C 180,E1 -11778.023,E2 -11778.023} C_VEL
LIN {X 0,Y 392.912,Z 707.625,A -85,B 0,C 180,E1 -11779.045,E2 -11779.045} C_VEL
LIN {X 0,Y 391.949,Z 717.91,A -85,B 0,C 180,E1 -11780.192,E2 -11780.192} C_VEL
LIN {X 0,Y 391.348,Z 725.851,A -85,B 0,C 180,E1 -11781.283,E2 -11781.283} C_VEL
LIN {X 0,Y 390.712,Z 733.327,A -85,B 0,C 180,E1 -11782.507,E2 -11782.507} C_VEL
LIN {X 0,Y 390.084,Z 741.08,A -85,B 0,C 180,E1 -11784.054,E2 -11784.054} C_VEL
LIN {X 0,Y 389.67,Z 746.347,A -85,B 0,C 180,E1 -11785.345,E2 -11785.345} C_VEL
LIN {X 0,Y 389.181,Z 751.497,A -85,B 0,C 180,E1 -11786.895,E2 -11786.895} C_VEL
LIN {X 0,Y 388.931,Z 755.495,A -85,B 0,C 180,E1 -11788.447,E2 -11788.447} C_VEL
LIN {X 0,Y 388.74,Z 758.459,A -85,B 0,C 180,E1 -11790,E2 -11790} C_VEL
LIN {X 0,Y 388.743,Z 759.904,A -85,B 0,C 180,E1 -11791.036,E2 -11791.036} C_VEL
LIN {X 0,Y 388.711,Z 760.925,A -85,B 0,C 180,E1 -11792.072,E2 -11792.072} C_VEL
LIN {X 0,Y 388.671,Z 761.824,A -85,B 0,C 180,E1 -11794.148,E2 -11794.148} C_VEL
LIN {X 0,Y 388.732,Z 761.223,A -85,B 0,C 180,E1 -11796.084,E2 -11796.084} C_VEL
LIN {X 0,Y 388.796,Z 760.166,A -85,B 0,C 180,E1 -11797.269,E2 -11797.269} C_VEL
LIN {X 0,Y 388.835,Z 758.826,A -85,B 0,C 180,E1 -11798.314,E2 -11798.314} C_VEL
LIN {X 0,Y 389,Z 755.779,A -85,B 0,C 180,E1 -11799.973,E2 -11799.973} C_VEL
LIN {X 0,Y 388.489,Z 753.931,A -85,B 0,C 180,E1 -11800.795,E2 -11800.795} C_VEL
LIN {X 0,Y 385.996,Z 750.506,A -85,B 0,C 180,E1 -11802.125,E2 -11802.125} C_VEL
LIN {X 0,Y 383.563,Z 746.486,A -85,B 0,C 180,E1 -11803.428,E2 -11803.428} C_VEL
LIN {X 0,Y 383.152,Z 743.575,A -85,B 0,C 180,E1 -11804.196,E2 -11804.196} C_VEL
LIN {X 0,Y 383.993,Z 735.586,A -85,B 0,C 180,E1 -11805.934,E2 -11805.934} C_VEL
LIN {X 0,Y 384.865,Z 728.01,A -85,B 0,C 180,E1 -11807.262,E2 -11807.262} C_VEL
LIN {X 0,Y 385.674,Z 719.673,A -85,B 0,C 180,E1 -11808.475,E2 -11808.475} C_VEL
LIN {X 0,Y 386.617,Z 709.82,A -85,B 0,C 180,E1 -11809.651,E2 -11809.651} C_VEL
LIN {X 0,Y 387.657,Z 698.7,A -85,B 0,C 180,E1 -11810.702,E2 -11810.702} C_VEL
LIN {X 0,Y 388.586,Z 687.209,A -85,B 0,C 180,E1 -11811.553,E2 -11811.553} C_VEL
LIN {X 0,Y 389.262,Z 674.216,A -85,B 0,C 180,E1 -11812.28,E2 -11812.28} C_VEL
LIN {X 0,Y 389.857,Z 660.575,A -85,B 0,C 180,E1 -11812.78,E2 -11812.78} C_VEL
LIN {X 0,Y 390.306,Z 637.763,A -85,B 0,C 180,E1 -11813.244,E2 -11813.244} C_VEL
LIN {X 0,Y 391.126,Z 574.613,A -85,B 0,C 180,E1 -11814.42,E2 -11814.42} C_VEL
LIN {X 0,Y 386.084,Z 552.565,A -85,B 0,C 180,E1 -11815.159,E2 -11815.159} C_VEL
LIN {X 0,Y 385.881,Z 551.403,A -85,B 0,C 180,E1 -11815.251,E2 -11815.251} C_VEL
LIN {X 0,Y 384.251,Z 542.284,A -85,B 0,C 180,E1 -11817.8,E2 -11817.8} C_VEL
LIN {X 0,Y 383.034,Z 536.775,A -85,B 0,C 180,E1 -11819.469,E2 -11819.469} C_VEL
LIN {X 0,Y 383.003,Z 536.777,A -85,B 0,C 180,E1 -11823.4,E2 -11823.4} C_VEL
LIN {X 0,Y 383.033,Z 536.774,A -85,B 0,C 180,E1 -11826.164,E2 -11826.164} C_VEL
LIN {X 0,Y 383.019,Z 536.774,A -85,B 0,C 180,E1 -11829.956,E2 -11829.956} C_VEL
LIN {X 0,Y 383.063,Z 536.77,A -85,B 0,C 180,E1 -11832.787,E2 -11832.787} C_VEL
LIN {X 0,Y 383.007,Z 536.773,A -85,B 0,C 180,E1 -11835.79,E2 -11835.79} C_VEL
LIN {X 0,Y 383.011,Z 536.766,A -85,B 0,C 180,E1 -11838.79,E2 -11838.79} C_VEL
LIN {X 0,Y 382.998,Z 536.776,A -85,B 0,C 180,E1 -11842.095,E2 -11842.095} C_VEL
LIN {X 0,Y 383.013,Z 536.772,A -85,B 0,C 180,E1 -11845.331,E2 -11845.331} C_VEL
LIN {X 0,Y 382.982,Z 536.774,A -85,B 0,C 180,E1 -11849.081,E2 -11849.081} C_VEL
LIN {X 0,Y 383.051,Z 536.768,A -85,B 0,C 180,E1 -11852.697,E2 -11852.697} C_VEL
LIN {X 0,Y 383.045,Z 536.771,A -85,B 0,C 180,E1 -11855.039,E2 -11855.039} C_VEL
LIN {X 0,Y 382.986,Z 536.774,A -85,B 0,C 180,E1 -11858.468,E2 -11858.468} C_VEL
LIN {X 0,Y 383.055,Z 536.764,A -85,B 0,C 180,E1 -11861.826,E2 -11861.826} C_VEL
LIN {X 0,Y 383.102,Z 536.762,A -85,B 0,C 180,E1 -11865.118,E2 -11865.118} C_VEL
LIN {X 0,Y 383.09,Z 536.761,A -85,B 0,C 180,E1 -11868.357,E2 -11868.357} C_VEL
LIN {X 0,Y 383.256,Z 536.739,A -85,B 0,C 180,E1 -11871.975,E2 -11871.975} C_VEL
LIN {X 0,Y 383.192,Z 536.756,A -85,B 0,C 180,E1 -11874.738,E2 -11874.738} C_VEL
LIN {X 0,Y 383.38,Z 536.72,A -85,B 0,C 180,E1 -11877.899,E2 -11877.899} C_VEL
LIN {X 0,Y 383.512,Z 536.71,A -85,B 0,C 180,E1 -11880,E2 -11880} C_VEL
LIN {X 0,Y 383.244,Z 536.738,A -85,B 0,C 180,E1 -11883.154,E2 -11883.154} C_VEL
LIN {X 0,Y 383.274,Z 536.743,A -85,B 0,C 180,E1 -11886.316,E2 -11886.316} C_VEL
LIN {X 0,Y 383.143,Z 536.753,A -85,B 0,C 180,E1 -11889.502,E2 -11889.502} C_VEL
LIN {X 0,Y 383.117,Z 536.752,A -85,B 0,C 180,E1 -11893.536,E2 -11893.536} C_VEL
LIN {X 0,Y 383.086,Z 536.761,A -85,B 0,C 180,E1 -11897.455,E2 -11897.455} C_VEL
LIN {X 0,Y 383.021,Z 536.777,A -85,B 0,C 180,E1 -11900.647,E2 -11900.647} C_VEL
LIN {X 0,Y 383.018,Z 536.768,A -85,B 0,C 180,E1 -11903.808,E2 -11903.808} C_VEL
LIN {X 0,Y 383.073,Z 536.767,A -85,B 0,C 180,E1 -11906.124,E2 -11906.124} C_VEL
LIN {X 0,Y 383.043,Z 536.77,A -85,B 0,C 180,E1 -11908.492,E2 -11908.492} C_VEL
LIN {X 0,Y 383.005,Z 536.776,A -85,B 0,C 180,E1 -11912.15,E2 -11912.15} C_VEL
LIN {X 0,Y 383.012,Z 536.778,A -85,B 0,C 180,E1 -11914.669,E2 -11914.669} C_VEL
LIN {X 0,Y 382.998,Z 536.775,A -85,B 0,C 180,E1 -11917.905,E2 -11917.905} C_VEL
LIN {X 0,Y 383.008,Z 536.775,A -85,B 0,C 180,E1 -11921.344,E2 -11921.344} C_VEL
LIN {X 0,Y 382.993,Z 536.78,A -85,B 0,C 180,E1 -11924.304,E2 -11924.304} C_VEL
LIN {X 0,Y 383.006,Z 536.776,A -85,B 0,C 180,E1 -11927.241,E2 -11927.241} C_VEL
LIN {X 0,Y 383.014,Z 536.778,A -85,B 0,C 180,E1 -11930.414,E2 -11930.414} C_VEL
LIN {X 0,Y 383.024,Z 536.774,A -85,B 0,C 180,E1 -11934.045,E2 -11934.045} C_VEL
LIN {X 0,Y 382.985,Z 536.779,A -85,B 0,C 180,E1 -11937.579,E2 -11937.579} C_VEL
LIN {X 0,Y 383.047,Z 536.804,A -85,B 0,C 180,E1 -11940.532,E2 -11940.532} C_VEL
LIN {X 0,Y 385.409,Z 547.648,A -85,B 0,C 180,E1 -11943.32,E2 -11943.32} C_VEL
LIN {X 0,Y 386.938,Z 555.713,A -85,B 0,C 180,E1 -11945.308,E2 -11945.308} C_VEL
LIN {X 0,Y 386.033,Z 566.653,A -85,B 0,C 180,E1 -11947.766,E2 -11947.766} C_VEL
LIN {X 0,Y 385.553,Z 571.386,A -85,B 0,C 180,E1 -11948.812,E2 -11948.812} C_VEL
LIN {X 0,Y 390.156,Z 596.684,A -85,B 0,C 180,E1 -11949.596,E2 -11949.596} C_VEL
LIN {X 0,Y 390.888,Z 603.157,A -85,B 0,C 180,E1 -11949.764,E2 -11949.764} C_VEL
LIN {X 0,Y 389.705,Z 679.467,A -85,B 0,C 180,E1 -11951.195,E2 -11951.195} C_VEL
LIN {X 0,Y 389.115,Z 692.74,A -85,B 0,C 180,E1 -11951.643,E2 -11951.643} C_VEL
LIN {X 0,Y 388.345,Z 704.334,A -85,B 0,C 180,E1 -11952.219,E2 -11952.219} C_VEL
LIN {X 0,Y 387.461,Z 715.914,A -85,B 0,C 180,E1 -11952.994,E2 -11952.994} C_VEL
LIN {X 0,Y 386.339,Z 727.789,A -85,B 0,C 180,E1 -11954.03,E2 -11954.03} C_VEL
LIN {X 0,Y 385.299,Z 738.391,A -85,B 0,C 180,E1 -11955.205,E2 -11955.205} C_VEL
LIN {X 0,Y 384.443,Z 747.955,A -85,B 0,C 180,E1 -11956.522,E2 -11956.522} C_VEL
LIN {X 0,Y 383.395,Z 757.176,A -85,B 0,C 180,E1 -11958.099,E2 -11958.099} C_VEL
LIN {X 0,Y 382.708,Z 764.596,A -85,B 0,C 180,E1 -11959.686,E2 -11959.686} C_VEL
LIN {X 0,Y 382.144,Z 771.45,A -85,B 0,C 180,E1 -11961.54,E2 -11961.54} C_VEL
LIN {X 0,Y 381.786,Z 775.978,A -85,B 0,C 180,E1 -11963.128,E2 -11963.128} C_VEL
LIN {X 0,Y 381.648,Z 779.428,A -85,B 0,C 180,E1 -11964.717,E2 -11964.717} C_VEL
LIN {X 0,Y 381.628,Z 781.152,A -85,B 0,C 180,E1 -11965.776,E2 -11965.776} C_VEL
LIN {X 0,Y 381.559,Z 783.394,A -85,B 0,C 180,E1 -11967.889,E2 -11967.889} C_VEL
LIN {X 0,Y 381.617,Z 783.92,A -85,B 0,C 180,E1 -11968.945,E2 -11968.945} C_VEL
LIN {X 0,Y 381.638,Z 784.014,A -85,B 0,C 180,E1 -11970,E2 -11970} C_VEL
LIN {X 0,Y 381.617,Z 783.72,A -85,B 0,C 180,E1 -11971.055,E2 -11971.055} C_VEL
LIN {X 0,Y 381.562,Z 783.039,A -85,B 0,C 180,E1 -11972.111,E2 -11972.111} C_VEL
LIN {X 0,Y 381.549,Z 781.96,A -85,B 0,C 180,E1 -11973.168,E2 -11973.168} C_VEL
LIN {X 0,Y 381.628,Z 780.428,A -85,B 0,C 180,E1 -11974.224,E2 -11974.224} C_VEL
LIN {X 0,Y 381.689,Z 776.608,A -85,B 0,C 180,E1 -11976.121,E2 -11976.121} C_VEL
LIN {X 0,Y 381.955,Z 771.557,A -85,B 0,C 180,E1 -11977.932,E2 -11977.932} C_VEL
LIN {X 0,Y 382.435,Z 764.687,A -85,B 0,C 180,E1 -11979.787,E2 -11979.787} C_VEL
LIN {X 0,Y 383,Z 757.224,A -85,B 0,C 180,E1 -11981.377,E2 -11981.377} C_VEL
LIN {X 0,Y 383.77,Z 749.621,A -85,B 0,C 180,E1 -11982.694,E2 -11982.694} C_VEL
LIN {X 0,Y 384.52,Z 740.975,A -85,B 0,C 180,E1 -11983.936,E2 -11983.936} C_VEL
LIN {X 0,Y 385.289,Z 731.418,A -85,B 0,C 180,E1 -11985.066,E2 -11985.066} C_VEL
LIN {X 0,Y 386.147,Z 720.343,A -85,B 0,C 180,E1 -11986.114,E2 -11986.114} C_VEL
LIN {X 0,Y 387.108,Z 707.929,A -85,B 0,C 180,E1 -11987.022,E2 -11987.022} C_VEL
LIN {X 0,Y 387.78,Z 696.128,A -85,B 0,C 180,E1 -11987.672,E2 -11987.672} C_VEL
LIN {X 0,Y 388.388,Z 683.35,A -85,B 0,C 180,E1 -11988.154,E2 -11988.154} C_VEL
LIN {X 0,Y 388.745,Z 666.994,A -85,B 0,C 180,E1 -11988.512,E2 -11988.512} C_VEL
LIN {X 0,Y 389.561,Z 601.212,A -85,B 0,C 180,E1 -11989.721,E2 -11989.721} C_VEL
LIN {X 0,Y 385.017,Z 571.464,A -85,B 0,C 180,E1 -11990.537,E2 -11990.537} C_VEL
LIN {X 0,Y 386.361,Z 555.207,A -85,B 0,C 180,E1 -11994.098,E2 -11994.098} C_VEL
LIN {X 0,Y 385.444,Z 548.54,A -85,B 0,C 180,E1 -11995.66,E2 -11995.66} C_VEL
LIN {X 0,Y 383.07,Z 536.769,A -85,B 0,C 180,E1 -11998.564,E2 -11998.564} C_VEL
LIN {X 0,Y 382.985,Z 536.775,A -85,B 0,C 180,E1 -12002.421,E2 -12002.421} C_VEL
LIN {X 0,Y 383.024,Z 536.772,A -85,B 0,C 180,E1 -12005.955,E2 -12005.955} C_VEL
LIN {X 0,Y 383.014,Z 536.777,A -85,B 0,C 180,E1 -12009.586,E2 -12009.586} C_VEL
LIN {X 0,Y 383.002,Z 536.773,A -85,B 0,C 180,E1 -12012.778,E2 -12012.778} C_VEL
LIN {X 0,Y 382.994,Z 536.777,A -85,B 0,C 180,E1 -12015.789,E2 -12015.789} C_VEL
LIN {X 0,Y 383.01,Z 536.772,A -85,B 0,C 180,E1 -12018.791,E2 -12018.791} C_VEL
LIN {X 0,Y 382.998,Z 536.774,A -85,B 0,C 180,E1 -12022.095,E2 -12022.095} C_VEL
LIN {X 0,Y 383.012,Z 536.777,A -85,B 0,C 180,E1 -12025.331,E2 -12025.331} C_VEL
LIN {X 0,Y 382.98,Z 536.778,A -85,B 0,C 180,E1 -12029.081,E2 -12029.081} C_VEL
LIN {X 0,Y 383.05,Z 536.767,A -85,B 0,C 180,E1 -12032.698,E2 -12032.698} C_VEL
LIN {X 0,Y 383.044,Z 536.77,A -85,B 0,C 180,E1 -12035.039,E2 -12035.039} C_VEL
LIN {X 0,Y 382.984,Z 536.775,A -85,B 0,C 180,E1 -12038.469,E2 -12038.469} C_VEL
LIN {X 0,Y 383.081,Z 536.766,A -85,B 0,C 180,E1 -12041.827,E2 -12041.827} C_VEL
LIN {X 0,Y 383.102,Z 536.763,A -85,B 0,C 180,E1 -12045.118,E2 -12045.118} C_VEL
LIN {X 0,Y 383.089,Z 536.762,A -85,B 0,C 180,E1 -12048.358,E2 -12048.358} C_VEL
LIN {X 0,Y 383.256,Z 536.742,A -85,B 0,C 180,E1 -12051.974,E2 -12051.974} C_VEL
LIN {X 0,Y 383.191,Z 536.75,A -85,B 0,C 180,E1 -12054.738,E2 -12054.738} C_VEL
LIN {X 0,Y 383.379,Z 536.728,A -85,B 0,C 180,E1 -12057.899,E2 -12057.899} C_VEL
LIN {X 0,Y 383.51,Z 536.711,A -85,B 0,C 180,E1 -12060,E2 -12060} C_VEL
LIN {X 0,Y 383.245,Z 536.746,A -85,B 0,C 180,E1 -12063.154,E2 -12063.154} C_VEL
LIN {X 0,Y 383.255,Z 536.741,A -85,B 0,C 180,E1 -12066.631,E2 -12066.631} C_VEL
LIN {X 0,Y 383.144,Z 536.761,A -85,B 0,C 180,E1 -12069.502,E2 -12069.502} C_VEL
LIN {X 0,Y 383.117,Z 536.764,A -85,B 0,C 180,E1 -12073.537,E2 -12073.537} C_VEL
LIN {X 0,Y 383.087,Z 536.769,A -85,B 0,C 180,E1 -12077.455,E2 -12077.455} C_VEL
LIN {X 0,Y 383.024,Z 536.77,A -85,B 0,C 180,E1 -12080.648,E2 -12080.648} C_VEL
LIN {X 0,Y 383.027,Z 536.772,A -85,B 0,C 180,E1 -12083.808,E2 -12083.808} C_VEL
LIN {X 0,Y 383.074,Z 536.764,A -85,B 0,C 180,E1 -12086.124,E2 -12086.124} C_VEL
LIN {X 0,Y 383.044,Z 536.767,A -85,B 0,C 180,E1 -12088.493,E2 -12088.493} C_VEL
LIN {X 0,Y 383.006,Z 536.773,A -85,B 0,C 180,E1 -12092.15,E2 -12092.15} C_VEL
LIN {X 0,Y 383.013,Z 536.772,A -85,B 0,C 180,E1 -12094.669,E2 -12094.669} C_VEL
LIN {X 0,Y 382.998,Z 536.775,A -85,B 0,C 180,E1 -12097.905,E2 -12097.905} C_VEL
LIN {X 0,Y 382.982,Z 536.781,A -85,B 0,C 180,E1 -12101.348,E2 -12101.348} C_VEL
LIN {X 0,Y 383.006,Z 536.772,A -85,B 0,C 180,E1 -12104.306,E2 -12104.306} C_VEL
LIN {X 0,Y 383.073,Z 536.769,A -85,B 0,C 180,E1 -12107.25,E2 -12107.25} C_VEL
LIN {X 0,Y 383.021,Z 536.77,A -85,B 0,C 180,E1 -12110.413,E2 -12110.413} C_VEL
LIN {X 0,Y 383.026,Z 536.771,A -85,B 0,C 180,E1 -12114.046,E2 -12114.046} C_VEL
LIN {X 0,Y 382.986,Z 536.779,A -85,B 0,C 180,E1 -12117.579,E2 -12117.579} C_VEL
LIN {X 0,Y 382.992,Z 536.774,A -85,B 0,C 180,E1 -12120.301,E2 -12120.301} C_VEL
LIN {X 0,Y 383.058,Z 536.766,A -85,B 0,C 180,E1 -12122.699,E2 -12122.699} C_VEL
LIN {X 0,Y 383.035,Z 536.769,A -85,B 0,C 180,E1 -12126.193,E2 -12126.193} C_VEL
LIN {X 0,Y 383.084,Z 536.861,A -85,B 0,C 180,E1 -12129.601,E2 -12129.601} C_VEL
LIN {X 0,Y 385.283,Z 548.336,A -85,B 0,C 180,E1 -12132.758,E2 -12132.758} C_VEL
LIN {X 0,Y 385.299,Z 551.486,A -85,B 0,C 180,E1 -12133.569,E2 -12133.569} C_VEL
LIN {X 0,Y 389.892,Z 575.144,A -85,B 0,C 180,E1 -12134.256,E2 -12134.256} C_VEL
LIN {X 0,Y 388.741,Z 658.372,A -85,B 0,C 180,E1 -12135.807,E2 -12135.807} C_VEL
LIN {X 0,Y 388.288,Z 670.783,A -85,B 0,C 180,E1 -12136.224,E2 -12136.224} C_VEL
LIN {X 0,Y 387.686,Z 683.058,A -85,B 0,C 180,E1 -12136.837,E2 -12136.837} C_VEL
LIN {X 0,Y 386.892,Z 695.43,A -85,B 0,C 180,E1 -12137.676,E2 -12137.676} C_VEL
LIN {X 0,Y 386.092,Z 707.01,A -85,B 0,C 180,E1 -12138.716,E2 -12138.716} C_VEL
LIN {X 0,Y 385.09,Z 717.436,A -85,B 0,C 180,E1 -12139.883,E2 -12139.883} C_VEL
LIN {X 0,Y 384.416,Z 725.383,A -85,B 0,C 180,E1 -12140.975,E2 -12140.975} C_VEL
LIN {X 0,Y 383.709,Z 733.799,A -85,B 0,C 180,E1 -12142.369,E2 -12142.369} C_VEL
LIN {X 0,Y 383.047,Z 741.486,A -85,B 0,C 180,E1 -12143.944,E2 -12143.944} C_VEL
LIN {X 0,Y 382.632,Z 746.731,A -85,B 0,C 180,E1 -12145.259,E2 -12145.259} C_VEL
LIN {X 0,Y 382.128,Z 751.839,A -85,B 0,C 180,E1 -12146.837,E2 -12146.837} C_VEL
LIN {X 0,Y 381.851,Z 755.807,A -85,B 0,C 180,E1 -12148.418,E2 -12148.418} C_VEL
LIN {X 0,Y 381.67,Z 758.744,A -85,B 0,C 180,E1 -12150,E2 -12150} C_VEL
LIN {X 0,Y 381.656,Z 760.159,A -85,B 0,C 180,E1 -12151.055,E2 -12151.055} C_VEL
LIN {X 0,Y 381.609,Z 761.166,A -85,B 0,C 180,E1 -12152.111,E2 -12152.111} C_VEL
LIN {X 0,Y 381.596,Z 762.036,A -85,B 0,C 180,E1 -12154.225,E2 -12154.225} C_VEL
LIN {X 0,Y 381.661,Z 761.48,A -85,B 0,C 180,E1 -12156.079,E2 -12156.079} C_VEL
LIN {X 0,Y 381.702,Z 760.32,A -85,B 0,C 180,E1 -12157.405,E2 -12157.405} C_VEL
LIN {X 0,Y 381.752,Z 758.965,A -85,B 0,C 180,E1 -12158.469,E2 -12158.469} C_VEL
LIN {X 0,Y 381.939,Z 756.091,A -85,B 0,C 180,E1 -12160.067,E2 -12160.067} C_VEL
LIN {X 0,Y 382.342,Z 752.179,A -85,B 0,C 180,E1 -12161.665,E2 -12161.665} C_VEL
LIN {X 0,Y 382.81,Z 746.879,A -85,B 0,C 180,E1 -12163.336,E2 -12163.336} C_VEL
LIN {X 0,Y 383.152,Z 743.575,A -85,B 0,C 180,E1 -12164.196,E2 -12164.196} C_VEL
LIN {X 0,Y 382.783,Z 740.492,A -85,B 0,C 180,E1 -12164.946,E2 -12164.946} C_VEL
LIN {X 0,Y 379.627,Z 732.927,A -85,B 0,C 180,E1 -12166.634,E2 -12166.634} C_VEL
LIN {X 0,Y 378.34,Z 728.034,A -85,B 0,C 180,E1 -12167.551,E2 -12167.551} C_VEL
LIN {X 0,Y 378.34,Z 725.335,A -85,B 0,C 180,E1 -12167.985,E2 -12167.985} C_VEL
LIN {X 0,Y 379.332,Z 715.42,A -85,B 0,C 180,E1 -12169.34,E2 -12169.34} C_VEL
LIN {X 0,Y 380.291,Z 705.68,A -85,B 0,C 180,E1 -12170.415,E2 -12170.415} C_VEL
LIN {X 0,Y 381.212,Z 695.109,A -85,B 0,C 180,E1 -12171.352,E2 -12171.352} C_VEL
LIN {X 0,Y 382.186,Z 682.345,A -85,B 0,C 180,E1 -12172.217,E2 -12172.217} C_VEL
LIN {X 0,Y 382.847,Z 670.344,A -85,B 0,C 180,E1 -12172.813,E2 -12172.813} C_VEL
LIN {X 0,Y 383.316,Z 657.845,A -85,B 0,C 180,E1 -12173.23,E2 -12173.23} C_VEL
LIN {X 0,Y 384.636,Z 576.056,A -85,B 0,C 180,E1 -12174.784,E2 -12174.784} C_VEL
LIN {X 0,Y 379.731,Z 554.517,A -85,B 0,C 180,E1 -12175.525,E2 -12175.525} C_VEL
LIN {X 0,Y 378.807,Z 551.696,A -85,B 0,C 180,E1 -12175.675,E2 -12175.675} C_VEL
LIN {X 0,Y 377.103,Z 542.747,A -85,B 0,C 180,E1 -12178.244,E2 -12178.244} C_VEL
LIN {X 0,Y 375.963,Z 537.652,A -85,B 0,C 180,E1 -12179.771,E2 -12179.771} C_VEL
LIN {X 0,Y 375.949,Z 537.656,A -85,B 0,C 180,E1 -12182.828,E2 -12182.828} C_VEL
LIN {X 0,Y 375.958,Z 537.653,A -85,B 0,C 180,E1 -12185.414,E2 -12185.414} C_VEL
LIN {X 0,Y 375.977,Z 537.649,A -85,B 0,C 180,E1 -12188.27,E2 -12188.27} C_VEL
LIN {X 0,Y 375.988,Z 537.648,A -85,B 0,C 180,E1 -12191.609,E2 -12191.609} C_VEL
LIN {X 0,Y 375.968,Z 537.651,A -85,B 0,C 180,E1 -12195.261,E2 -12195.261} C_VEL
LIN {X 0,Y 375.977,Z 537.641,A -85,B 0,C 180,E1 -12199.137,E2 -12199.137} C_VEL
LIN {X 0,Y 375.963,Z 537.652,A -85,B 0,C 180,E1 -12201.911,E2 -12201.911} C_VEL
LIN {X 0,Y 375.975,Z 537.648,A -85,B 0,C 180,E1 -12205.332,E2 -12205.332} C_VEL
LIN {X 0,Y 375.955,Z 537.656,A -85,B 0,C 180,E1 -12208.437,E2 -12208.437} C_VEL
LIN {X 0,Y 375.997,Z 537.648,A -85,B 0,C 180,E1 -12212.141,E2 -12212.141} C_VEL
LIN {X 0,Y 376,Z 537.647,A -85,B 0,C 180,E1 -12214.538,E2 -12214.538} C_VEL
LIN {X 0,Y 375.956,Z 537.646,A -85,B 0,C 180,E1 -12218.045,E2 -12218.045} C_VEL
LIN {X 0,Y 376.001,Z 537.642,A -85,B 0,C 180,E1 -12221.473,E2 -12221.473} C_VEL
LIN {X 0,Y 376.05,Z 537.643,A -85,B 0,C 180,E1 -12224.832,E2 -12224.832} C_VEL
LIN {X 0,Y 376.042,Z 537.636,A -85,B 0,C 180,E1 -12228.136,E2 -12228.136} C_VEL
LIN {X 0,Y 376.211,Z 537.616,A -85,B 0,C 180,E1 -12231.918,E2 -12231.918} C_VEL
LIN {X 0,Y 376.164,Z 537.63,A -85,B 0,C 180,E1 -12234.64,E2 -12234.64} C_VEL
LIN {X 0,Y 376.346,Z 537.596,A -85,B 0,C 180,E1 -12237.859,E2 -12237.859} C_VEL
LIN {X 0,Y 376.482,Z 537.586,A -85,B 0,C 180,E1 -12240,E2 -12240} C_VEL
LIN {X 0,Y 376.182,Z 537.618,A -85,B 0,C 180,E1 -12243.213,E2 -12243.213} C_VEL
LIN {X 0,Y 376.232,Z 537.622,A -85,B 0,C 180,E1 -12246.435,E2 -12246.435} C_VEL
LIN {X 0,Y 376.111,Z 537.629,A -85,B 0,C 180,E1 -12249.682,E2 -12249.682} C_VEL
LIN {X 0,Y 376.081,Z 537.628,A -85,B 0,C 180,E1 -12253.658,E2 -12253.658} C_VEL
LIN {X 0,Y 376.036,Z 537.639,A -85,B 0,C 180,E1 -12257.607,E2 -12257.607} C_VEL
LIN {X 0,Y 375.971,Z 537.653,A -85,B 0,C 180,E1 -12260.832,E2 -12260.832} C_VEL
LIN {X 0,Y 375.982,Z 537.648,A -85,B 0,C 180,E1 -12264.282,E2 -12264.282} C_VEL
LIN {X 0,Y 376.013,Z 537.643,A -85,B 0,C 180,E1 -12266.653,E2 -12266.653} C_VEL
LIN {X 0,Y 375.97,Z 537.651,A -85,B 0,C 180,E1 -12269.079,E2 -12269.079} C_VEL
LIN {X 0,Y 375.943,Z 537.657,A -85,B 0,C 180,E1 -12272.829,E2 -12272.829} C_VEL
LIN {X 0,Y 375.953,Z 537.652,A -85,B 0,C 180,E1 -12275.416,E2 -12275.416} C_VEL
LIN {X 0,Y 375.973,Z 537.653,A -85,B 0,C 180,E1 -12278.272,E2 -12278.272} C_VEL
LIN {X 0,Y 375.955,Z 537.653,A -85,B 0,C 180,E1 -12281.606,E2 -12281.606} C_VEL
LIN {X 0,Y 375.924,Z 537.657,A -85,B 0,C 180,E1 -12285.269,E2 -12285.269} C_VEL
LIN {X 0,Y 375.932,Z 537.659,A -85,B 0,C 180,E1 -12288.4,E2 -12288.4} C_VEL
LIN {X 0,Y 375.973,Z 537.651,A -85,B 0,C 180,E1 -12291.73,E2 -12291.73} C_VEL
LIN {X 0,Y 375.978,Z 537.651,A -85,B 0,C 180,E1 -12295.333,E2 -12295.333} C_VEL
LIN {X 0,Y 375.956,Z 537.657,A -85,B 0,C 180,E1 -12298.439,E2 -12298.439} C_VEL
LIN {X 0,Y 375.993,Z 537.703,A -85,B 0,C 180,E1 -12300.155,E2 -12300.155} C_VEL
LIN {X 0,Y 378.434,Z 548.706,A -85,B 0,C 180,E1 -12303.053,E2 -12303.053} C_VEL
LIN {X 0,Y 379.936,Z 556.467,A -85,B 0,C 180,E1 -12305.012,E2 -12305.012} C_VEL
LIN {X 0,Y 379.815,Z 560.602,A -85,B 0,C 180,E1 -12305.979,E2 -12305.979} C_VEL
LIN {X 0,Y 378.731,Z 571.193,A -85,B 0,C 180,E1 -12308.382,E2 -12308.382} C_VEL
LIN {X 0,Y 383.551,Z 597.481,A -85,B 0,C 180,E1 -12309.218,E2 -12309.218} C_VEL
LIN {X 0,Y 384.283,Z 603.822,A -85,B 0,C 180,E1 -12309.387,E2 -12309.387} C_VEL
LIN {X 0,Y 383.009,Z 680.237,A -85,B 0,C 180,E1 -12310.853,E2 -12310.853} C_VEL
LIN {X 0,Y 382.342,Z 693.946,A -85,B 0,C 180,E1 -12311.34,E2 -12311.34} C_VEL
LIN {X 0,Y 381.613,Z 704.61,A -85,B 0,C 180,E1 -12311.894,E2 -12311.894} C_VEL
LIN {X 0,Y 380.697,Z 716.083,A -85,B 0,C 180,E1 -12312.682,E2 -12312.682} C_VEL
LIN {X 0,Y 379.514,Z 727.859,A -85,B 0,C 180,E1 -12313.735,E2 -12313.735} C_VEL
LIN {X 0,Y 378.4,Z 738.738,A -85,B 0,C 180,E1 -12314.971,E2 -12314.971} C_VEL
LIN {X 0,Y 377.531,Z 747.937,A -85,B 0,C 180,E1 -12316.27,E2 -12316.27} C_VEL
LIN {X 0,Y 376.437,Z 757.113,A -85,B 0,C 180,E1 -12317.876,E2 -12317.876} C_VEL
LIN {X 0,Y 375.71,Z 764.507,A -85,B 0,C 180,E1 -12319.492,E2 -12319.492} C_VEL
LIN {X 0,Y 375.082,Z 771.329,A -85,B 0,C 180,E1 -12321.379,E2 -12321.379} C_VEL
LIN {X 0,Y 374.727,Z 775.837,A -85,B 0,C 180,E1 -12322.998,E2 -12322.998} C_VEL
LIN {X 0,Y 374.555,Z 779.271,A -85,B 0,C 180,E1 -12324.617,E2 -12324.617} C_VEL
LIN {X 0,Y 374.554,Z 780.984,A -85,B 0,C 180,E1 -12325.696,E2 -12325.696} C_VEL
LIN {X 0,Y 374.458,Z 783.21,A -85,B 0,C 180,E1 -12327.849,E2 -12327.849} C_VEL
LIN {X 0,Y 374.517,Z 783.721,A -85,B 0,C 180,E1 -12328.925,E2 -12328.925} C_VEL
LIN {X 0,Y 374.554,Z 783.806,A -85,B 0,C 180,E1 -12330,E2 -12330} C_VEL
LIN {X 0,Y 374.517,Z 783.503,A -85,B 0,C 180,E1 -12331.075,E2 -12331.075} C_VEL
LIN {X 0,Y 374.461,Z 782.814,A -85,B 0,C 180,E1 -12332.151,E2 -12332.151} C_VEL
LIN {X 0,Y 374.464,Z 781.721,A -85,B 0,C 180,E1 -12333.228,E2 -12333.228} C_VEL
LIN {X 0,Y 374.554,Z 780.177,A -85,B 0,C 180,E1 -12334.304,E2 -12334.304} C_VEL
LIN {X 0,Y 374.584,Z 776.729,A -85,B 0,C 180,E1 -12336.069,E2 -12336.069} C_VEL
LIN {X 0,Y 374.892,Z 771.266,A -85,B 0,C 180,E1 -12338.082,E2 -12338.082} C_VEL
LIN {X 0,Y 375.408,Z 764.365,A -85,B 0,C 180,E1 -12339.972,E2 -12339.972} C_VEL
LIN {X 0,Y 376.007,Z 756.876,A -85,B 0,C 180,E1 -12341.591,E2 -12341.591} C_VEL
LIN {X 0,Y 376.801,Z 749.244,A -85,B 0,C 180,E1 -12342.933,E2 -12342.933} C_VEL
LIN {X 0,Y 377.722,Z 739.547,A -85,B 0,C 180,E1 -12344.329,E2 -12344.329} C_VEL
LIN {X 0,Y 378.609,Z 728.362,A -85,B 0,C 180,E1 -12345.614,E2 -12345.614} C_VEL
LIN {X 0,Y 379.566,Z 716.613,A -85,B 0,C 180,E1 -12346.678,E2 -12346.678} C_VEL
LIN {X 0,Y 380.409,Z 705.176,A -85,B 0,C 180,E1 -12347.47,E2 -12347.47} C_VEL
LIN {X 0,Y 381.135,Z 692.283,A -85,B 0,C 180,E1 -12348.129,E2 -12348.129} C_VEL
LIN {X 0,Y 381.687,Z 679.881,A -85,B 0,C 180,E1 -12348.554,E2 -12348.554} C_VEL
LIN {X 0,Y 382.721,Z 601.225,A -85,B 0,C 180,E1 -12350.054,E2 -12350.054} C_VEL
LIN {X 0,Y 378.075,Z 571.303,A -85,B 0,C 180,E1 -12350.89,E2 -12350.89} C_VEL
LIN {X 0,Y 379.313,Z 557.131,A -85,B 0,C 180,E1 -12354.055,E2 -12354.055} C_VEL
LIN {X 0,Y 379.146,Z 553.393,A -85,B 0,C 180,E1 -12354.922,E2 -12354.922} C_VEL
LIN {X 0,Y 376.886,Z 541.768,A -85,B 0,C 180,E1 -12357.786,E2 -12357.786} C_VEL
LIN {X 0,Y 376.027,Z 537.648,A -85,B 0,C 180,E1 -12358.837,E2 -12358.837} C_VEL
LIN {X 0,Y 375.947,Z 537.652,A -85,B 0,C 180,E1 -12362.828,E2 -12362.828} C_VEL
LIN {X 0,Y 375.956,Z 537.657,A -85,B 0,C 180,E1 -12365.415,E2 -12365.415} C_VEL
LIN {X 0,Y 375.973,Z 537.648,A -85,B 0,C 180,E1 -12368.27,E2 -12368.27} C_VEL
LIN {X 0,Y 375.933,Z 537.659,A -85,B 0,C 180,E1 -12371.6,E2 -12371.6} C_VEL
LIN {X 0,Y 375.95,Z 537.656,A -85,B 0,C 180,E1 -12375.264,E2 -12375.264} C_VEL
LIN {X 0,Y 375.976,Z 537.651,A -85,B 0,C 180,E1 -12379.138,E2 -12379.138} C_VEL
LIN {X 0,Y 375.963,Z 537.652,A -85,B 0,C 180,E1 -12381.911,E2 -12381.911} C_VEL
LIN {X 0,Y 375.974,Z 537.654,A -85,B 0,C 180,E1 -12385.332,E2 -12385.332} C_VEL
LIN {X 0,Y 375.953,Z 537.651,A -85,B 0,C 180,E1 -12388.438,E2 -12388.438} C_VEL
LIN {X 0,Y 375.995,Z 537.646,A -85,B 0,C 180,E1 -12392.141,E2 -12392.141} C_VEL
LIN {X 0,Y 375.998,Z 537.645,A -85,B 0,C 180,E1 -12394.538,E2 -12394.538} C_VEL
LIN {X 0,Y 375.95,Z 537.652,A -85,B 0,C 180,E1 -12398.045,E2 -12398.045} C_VEL
LIN {X 0,Y 376.016,Z 537.65,A -85,B 0,C 180,E1 -12401.474,E2 -12401.474} C_VEL
LIN {X 0,Y 376.05,Z 537.64,A -85,B 0,C 180,E1 -12404.832,E2 -12404.832} C_VEL
LIN {X 0,Y 376.042,Z 537.64,A -85,B 0,C 180,E1 -12408.136,E2 -12408.136} C_VEL
LIN {X 0,Y 376.212,Z 537.62,A -85,B 0,C 180,E1 -12411.917,E2 -12411.917} C_VEL
LIN {X 0,Y 376.163,Z 537.625,A -85,B 0,C 180,E1 -12414.64,E2 -12414.64} C_VEL
LIN {X 0,Y 376.345,Z 537.604,A -85,B 0,C 180,E1 -12417.86,E2 -12417.86} C_VEL
LIN {X 0,Y 376.48,Z 537.586,A -85,B 0,C 180,E1 -12420,E2 -12420} C_VEL
LIN {X 0,Y 376.183,Z 537.626,A -85,B 0,C 180,E1 -12423.213,E2 -12423.213} C_VEL
LIN {X 0,Y 376.22,Z 537.617,A -85,B 0,C 180,E1 -12426.619,E2 -12426.619} C_VEL
LIN {X 0,Y 376.111,Z 537.635,A -85,B 0,C 180,E1 -12429.682,E2 -12429.682} C_VEL
LIN {X 0,Y 376.082,Z 537.639,A -85,B 0,C 180,E1 -12433.658,E2 -12433.658} C_VEL
LIN {X 0,Y 376.036,Z 537.645,A -85,B 0,C 180,E1 -12437.607,E2 -12437.607} C_VEL
LIN {X 0,Y 375.971,Z 537.65,A -85,B 0,C 180,E1 -12440.833,E2 -12440.833} C_VEL
LIN {X 0,Y 375.987,Z 537.647,A -85,B 0,C 180,E1 -12444.282,E2 -12444.282} C_VEL
LIN {X 0,Y 376.014,Z 537.644,A -85,B 0,C 180,E1 -12446.653,E2 -12446.653} C_VEL
LIN {X 0,Y 375.971,Z 537.652,A -85,B 0,C 180,E1 -12449.079,E2 -12449.079} C_VEL
LIN {X 0,Y 375.945,Z 537.653,A -85,B 0,C 180,E1 -12452.829,E2 -12452.829} C_VEL
LIN {X 0,Y 375.953,Z 537.658,A -85,B 0,C 180,E1 -12455.416,E2 -12455.416} C_VEL
LIN {X 0,Y 375.972,Z 537.648,A -85,B 0,C 180,E1 -12458.272,E2 -12458.272} C_VEL
LIN {X 0,Y 375.932,Z 537.658,A -85,B 0,C 180,E1 -12461.602,E2 -12461.602} C_VEL
LIN {X 0,Y 375.977,Z 537.653,A -85,B 0,C 180,E1 -12465.261,E2 -12465.261} C_VEL
LIN {X 0,Y 375.988,Z 537.646,A -85,B 0,C 180,E1 -12468.391,E2 -12468.391} C_VEL
LIN {X 0,Y 375.967,Z 537.651,A -85,B 0,C 180,E1 -12471.913,E2 -12471.913} C_VEL
LIN {X 0,Y 375.979,Z 537.654,A -85,B 0,C 180,E1 -12475.334,E2 -12475.334} C_VEL
LIN {X 0,Y 375.958,Z 537.65,A -85,B 0,C 180,E1 -12478.439,E2 -12478.439} C_VEL
LIN {X 0,Y 375.997,Z 537.646,A -85,B 0,C 180,E1 -12482.142,E2 -12482.142} C_VEL
LIN {X 0,Y 376.008,Z 537.644,A -85,B 0,C 180,E1 -12484.54,E2 -12484.54} C_VEL
LIN {X 0,Y 375.965,Z 537.657,A -85,B 0,C 180,E1 -12488.046,E2 -12488.046} C_VEL
LIN {X 0,Y 376.012,Z 537.777,A -85,B 0,C 180,E1 -12489.346,E2 -12489.346} C_VEL
LIN {X 0,Y 377.992,Z 547.86,A -85,B 0,C 180,E1 -12492.181,E2 -12492.181} C_VEL
LIN {X 0,Y 378.405,Z 551.806,A -85,B 0,C 180,E1 -12493.214,E2 -12493.214} C_VEL
LIN {X 0,Y 383.145,Z 576.176,A -85,B 0,C 180,E1 -12493.938,E2 -12493.938} C_VEL
LIN {X 0,Y 381.951,Z 659.057,A -85,B 0,C 180,E1 -12495.515,E2 -12495.515} C_VEL
LIN {X 0,Y 381.447,Z 672.065,A -85,B 0,C 180,E1 -12495.972,E2 -12495.972} C_VEL
LIN {X 0,Y 380.833,Z 684.061,A -85,B 0,C 180,E1 -12496.595,E2 -12496.595} C_VEL
LIN {X 0,Y 380.006,Z 696.199,A -85,B 0,C 180,E1 -12497.449,E2 -12497.449} C_VEL
LIN {X 0,Y 379.176,Z 707.673,A -85,B 0,C 180,E1 -12498.507,E2 -12498.507} C_VEL
LIN {X 0,Y 378.135,Z 718.021,A -85,B 0,C 180,E1 -12499.695,E2 -12499.695} C_VEL
LIN {X 0,Y 377.433,Z 725.905,A -85,B 0,C 180,E1 -12500.807,E2 -12500.807} C_VEL
LIN {X 0,Y 376.709,Z 734.267,A -85,B 0,C 180,E1 -12502.227,E2 -12502.227} C_VEL
LIN {X 0,Y 376.012,Z 741.89,A -85,B 0,C 180,E1 -12503.831,E2 -12503.831} C_VEL
LIN {X 0,Y 375.579,Z 747.108,A -85,B 0,C 180,E1 -12505.17,E2 -12505.17} C_VEL
LIN {X 0,Y 375.058,Z 752.176,A -85,B 0,C 180,E1 -12506.777,E2 -12506.777} C_VEL
LIN {X 0,Y 374.775,Z 756.113,A -85,B 0,C 180,E1 -12508.388,E2 -12508.388} C_VEL
LIN {X 0,Y 374.602,Z 759.024,A -85,B 0,C 180,E1 -12510,E2 -12510} C_VEL
LIN {X 0,Y 374.571,Z 760.414,A -85,B 0,C 180,E1 -12511.075,E2 -12511.075} C_VEL
LIN {X 0,Y 374.474,Z 762.018,A -85,B 0,C 180,E1 -12513.228,E2 -12513.228} C_VEL
LIN {X 0,Y 374.522,Z 762.244,A -85,B 0,C 180,E1 -12514.305,E2 -12514.305} C_VEL
LIN {X 0,Y 374.566,Z 761.452,A -85,B 0,C 180,E1 -12516.464,E2 -12516.464} C_VEL
LIN {X 0,Y 374.619,Z 760.475,A -85,B 0,C 180,E1 -12517.546,E2 -12517.546} C_VEL
LIN {X 0,Y 374.685,Z 759.101,A -85,B 0,C 180,E1 -12518.63,E2 -12518.63} C_VEL
LIN {X 0,Y 374.902,Z 756.2,A -85,B 0,C 180,E1 -12520.258,E2 -12520.258} C_VEL
LIN {X 0,Y 375.33,Z 752.256,A -85,B 0,C 180,E1 -12521.886,E2 -12521.886} C_VEL
LIN {X 0,Y 375.9,Z 746.253,A -85,B 0,C 180,E1 -12523.765,E2 -12523.765} C_VEL
LIN {X 0,Y 376.671,Z 739.478,A -85,B 0,C 180,E1 -12525.419,E2 -12525.419} C_VEL
LIN {X 0,Y 377.62,Z 731.167,A -85,B 0,C 180,E1 -12527.045,E2 -12527.045} C_VEL
LIN {X 0,Y 378.34,Z 725.335,A -85,B 0,C 180,E1 -12527.985,E2 -12527.985} C_VEL
LIN {X 0,Y 378.129,Z 721.198,A -85,B 0,C 180,E1 -12528.619,E2 -12528.619} C_VEL
LIN {X 0,Y 376.048,Z 714.281,A -85,B 0,C 180,E1 -12529.651,E2 -12529.651} C_VEL
LIN {X 0,Y 374.033,Z 706.922,A -85,B 0,C 180,E1 -12530.61,E2 -12530.61} C_VEL
LIN {X 0,Y 373.915,Z 702.008,A -85,B 0,C 180,E1 -12531.122,E2 -12531.122} C_VEL
LIN {X 0,Y 374.899,Z 691.138,A -85,B 0,C 180,E1 -12532.019,E2 -12532.019} C_VEL
LIN {X 0,Y 375.731,Z 679.364,A -85,B 0,C 180,E1 -12532.765,E2 -12532.765} C_VEL
LIN {X 0,Y 376.38,Z 667.237,A -85,B 0,C 180,E1 -12533.317,E2 -12533.317} C_VEL
LIN {X 0,Y 376.796,Z 653.911,A -85,B 0,C 180,E1 -12533.704,E2 -12533.704} C_VEL
LIN {X 0,Y 377.999,Z 576.952,A -85,B 0,C 180,E1 -12535.183,E2 -12535.183} C_VEL
LIN {X 0,Y 373.672,Z 557.571,A -85,B 0,C 180,E1 -12535.862,E2 -12535.862} C_VEL
LIN {X 0,Y 371.671,Z 551.918,A -85,B 0,C 180,E1 -12536.149,E2 -12536.149} C_VEL
LIN {X 0,Y 369.742,Z 542.133,A -85,B 0,C 180,E1 -12539.03,E2 -12539.03} C_VEL
LIN {X 0,Y 368.942,Z 538.522,A -85,B 0,C 180,E1 -12540.159,E2 -12540.159} C_VEL
LIN {X 0,Y 368.896,Z 538.535,A -85,B 0,C 180,E1 -12543.537,E2 -12543.537} C_VEL
LIN {X 0,Y 368.902,Z 538.534,A -85,B 0,C 180,E1 -12546.855,E2 -12546.855} C_VEL
LIN {X 0,Y 368.951,Z 538.528,A -85,B 0,C 180,E1 -12550.364,E2 -12550.364} C_VEL
LIN {X 0,Y 368.954,Z 538.524,A -85,B 0,C 180,E1 -12553.627,E2 -12553.627} C_VEL
LIN {X 0,Y 368.905,Z 538.535,A -85,B 0,C 180,E1 -12556.698,E2 -12556.698} C_VEL
LIN {X 0,Y 368.949,Z 538.518,A -85,B 0,C 180,E1 -12559.635,E2 -12559.635} C_VEL
LIN {X 0,Y 368.899,Z 538.531,A -85,B 0,C 180,E1 -12563.143,E2 -12563.143} C_VEL
LIN {X 0,Y 368.892,Z 538.532,A -85,B 0,C 180,E1 -12566.461,E2 -12566.461} C_VEL
LIN {X 0,Y 368.918,Z 538.526,A -85,B 0,C 180,E1 -12570.31,E2 -12570.31} C_VEL
LIN {X 0,Y 368.976,Z 538.516,A -85,B 0,C 180,E1 -12573.534,E2 -12573.534} C_VEL
LIN {X 0,Y 368.96,Z 538.527,A -85,B 0,C 180,E1 -12576.421,E2 -12576.421} C_VEL
LIN {X 0,Y 368.929,Z 538.528,A -85,B 0,C 180,E1 -12579.946,E2 -12579.946} C_VEL
LIN {X 0,Y 368.968,Z 538.521,A -85,B 0,C 180,E1 -12583.398,E2 -12583.398} C_VEL
LIN {X 0,Y 369.05,Z 538.508,A -85,B 0,C 180,E1 -12586.79,E2 -12586.79} C_VEL
LIN {X 0,Y 369.06,Z 538.513,A -85,B 0,C 180,E1 -12590.131,E2 -12590.131} C_VEL
LIN {X 0,Y 369.193,Z 538.491,A -85,B 0,C 180,E1 -12593.441,E2 -12593.441} C_VEL
LIN {X 0,Y 369.311,Z 538.472,A -85,B 0,C 180,E1 -12597.819,E2 -12597.819} C_VEL
LIN {X 0,Y 369.451,Z 538.462,A -85,B 0,C 180,E1 -12600,E2 -12600} C_VEL
LIN {X 0,Y 369.31,Z 538.48,A -85,B 0,C 180,E1 -12602.181,E2 -12602.181} C_VEL
LIN {X 0,Y 369.192,Z 538.498,A -85,B 0,C 180,E1 -12606.558,E2 -12606.558} C_VEL
LIN {X 0,Y 369.059,Z 538.508,A -85,B 0,C 180,E1 -12609.868,E2 -12609.868} C_VEL
LIN {X 0,Y 369.029,Z 538.507,A -85,B 0,C 180,E1 -12613.772,E2 -12613.772} C_VEL
LIN {X 0,Y 368.994,Z 538.516,A -85,B 0,C 180,E1 -12617.769,E2 -12617.769} C_VEL
LIN {X 0,Y 368.902,Z 538.53,A -85,B 0,C 180,E1 -12621.221,E2 -12621.221} C_VEL
LIN {X 0,Y 368.948,Z 538.529,A -85,B 0,C 180,E1 -12624.776,E2 -12624.776} C_VEL
LIN {X 0,Y 368.964,Z 538.518,A -85,B 0,C 180,E1 -12627.203,E2 -12627.203} C_VEL
LIN {X 0,Y 368.917,Z 538.528,A -85,B 0,C 180,E1 -12629.69,E2 -12629.69} C_VEL
LIN {X 0,Y 368.891,Z 538.532,A -85,B 0,C 180,E1 -12633.539,E2 -12633.539} C_VEL
LIN {X 0,Y 368.898,Z 538.534,A -85,B 0,C 180,E1 -12636.857,E2 -12636.857} C_VEL
LIN {X 0,Y 368.948,Z 538.529,A -85,B 0,C 180,E1 -12640.365,E2 -12640.365} C_VEL
LIN {X 0,Y 368.89,Z 538.534,A -85,B 0,C 180,E1 -12643.619,E2 -12643.619} C_VEL
LIN {X 0,Y 368.883,Z 538.538,A -85,B 0,C 180,E1 -12646.697,E2 -12646.697} C_VEL
LIN {X 0,Y 368.91,Z 538.53,A -85,B 0,C 180,E1 -12649.644,E2 -12649.644} C_VEL
LIN {X 0,Y 368.9,Z 538.534,A -85,B 0,C 180,E1 -12653.145,E2 -12653.145} C_VEL
LIN {X 0,Y 368.895,Z 538.534,A -85,B 0,C 180,E1 -12656.463,E2 -12656.463} C_VEL
LIN {X 0,Y 368.934,Z 538.597,A -85,B 0,C 180,E1 -12659.761,E2 -12659.761} C_VEL
LIN {X 0,Y 371.479,Z 549.743,A -85,B 0,C 180,E1 -12662.772,E2 -12662.772} C_VEL
LIN {X 0,Y 373.104,Z 558.99,A -85,B 0,C 180,E1 -12665.145,E2 -12665.145} C_VEL
LIN {X 0,Y 371.985,Z 570.727,A -85,B 0,C 180,E1 -12667.874,E2 -12667.874} C_VEL
LIN {X 0,Y 371.971,Z 571.314,A -85,B 0,C 180,E1 -12667.951,E2 -12667.951} C_VEL
LIN {X 0,Y 376.805,Z 597.208,A -85,B 0,C 180,E1 -12668.794,E2 -12668.794} C_VEL
LIN {X 0,Y 377.72,Z 603.76,A -85,B 0,C 180,E1 -12668.984,E2 -12668.984} C_VEL
LIN {X 0,Y 376.4,Z 679.884,A -85,B 0,C 180,E1 -12670.468,E2 -12670.468} C_VEL
LIN {X 0,Y 375.718,Z 693.641,A -85,B 0,C 180,E1 -12670.964,E2 -12670.964} C_VEL
LIN {X 0,Y 374.893,Z 704.895,A -85,B 0,C 180,E1 -12671.558,E2 -12671.558} C_VEL
LIN {X 0,Y 373.924,Z 716.246,A -85,B 0,C 180,E1 -12672.358,E2 -12672.358} C_VEL
LIN {X 0,Y 372.7,Z 727.933,A -85,B 0,C 180,E1 -12673.429,E2 -12673.429} C_VEL
LIN {X 0,Y 371.565,Z 738.437,A -85,B 0,C 180,E1 -12674.645,E2 -12674.645} C_VEL
LIN {X 0,Y 370.611,Z 747.918,A -85,B 0,C 180,E1 -12676.009,E2 -12676.009} C_VEL
LIN {X 0,Y 369.493,Z 757.052,A -85,B 0,C 180,E1 -12677.644,E2 -12677.644} C_VEL
LIN {X 0,Y 368.707,Z 764.421,A -85,B 0,C 180,E1 -12679.29,E2 -12679.29} C_VEL
LIN {X 0,Y 368.041,Z 771.209,A -85,B 0,C 180,E1 -12681.213,E2 -12681.213} C_VEL
LIN {X 0,Y 367.667,Z 775.698,A -85,B 0,C 180,E1 -12682.863,E2 -12682.863} C_VEL
LIN {X 0,Y 367.467,Z 779.114,A -85,B 0,C 180,E1 -12684.513,E2 -12684.513} C_VEL
LIN {X 0,Y 367.459,Z 780.817,A -85,B 0,C 180,E1 -12685.612,E2 -12685.612} C_VEL
LIN {X 0,Y 367.359,Z 783.026,A -85,B 0,C 180,E1 -12687.807,E2 -12687.807} C_VEL
LIN {X 0,Y 367.416,Z 783.52,A -85,B 0,C 180,E1 -12688.904,E2 -12688.904} C_VEL
LIN {X 0,Y 367.456,Z 783.597,A -85,B 0,C 180,E1 -12690,E2 -12690} C_VEL
LIN {X 0,Y 367.417,Z 783.286,A -85,B 0,C 180,E1 -12691.096,E2 -12691.096} C_VEL
LIN {X 0,Y 367.362,Z 782.588,A -85,B 0,C 180,E1 -12692.193,E2 -12692.193} C_VEL
LIN {X 0,Y 367.382,Z 781.479,A -85,B 0,C 180,E1 -12693.29,E2 -12693.29} C_VEL
LIN {X 0,Y 367.459,Z 779.925,A -85,B 0,C 180,E1 -12694.388,E2 -12694.388} C_VEL
LIN {X 0,Y 367.482,Z 776.842,A -85,B 0,C 180,E1 -12696.017,E2 -12696.017} C_VEL
LIN {X 0,Y 367.722,Z 772.602,A -85,B 0,C 180,E1 -12697.688,E2 -12697.688} C_VEL
LIN {X 0,Y 368.188,Z 766.21,A -85,B 0,C 180,E1 -12699.614,E2 -12699.614} C_VEL
LIN {X 0,Y 368.775,Z 759.24,A -85,B 0,C 180,E1 -12701.264,E2 -12701.264} C_VEL
LIN {X 0,Y 369.685,Z 750.502,A -85,B 0,C 180,E1 -12702.907,E2 -12702.907} C_VEL
LIN {X 0,Y 370.551,Z 741.544,A -85,B 0,C 180,E1 -12704.274,E2 -12704.274} C_VEL
LIN {X 0,Y 371.505,Z 730.476,A -85,B 0,C 180,E1 -12705.639,E2 -12705.639} C_VEL
LIN {X 0,Y 372.448,Z 719.254,A -85,B 0,C 180,E1 -12706.724,E2 -12706.724} C_VEL
LIN {X 0,Y 373.476,Z 706.663,A -85,B 0,C 180,E1 -12707.664,E2 -12707.664} C_VEL
LIN {X 0,Y 374.226,Z 694.479,A -85,B 0,C 180,E1 -12708.334,E2 -12708.334} C_VEL
LIN {X 0,Y 374.881,Z 680.978,A -85,B 0,C 180,E1 -12708.832,E2 -12708.832} C_VEL
LIN {X 0,Y 375.289,Z 656.28,A -85,B 0,C 180,E1 -12709.343,E2 -12709.343} C_VEL
LIN {X 0,Y 376.025,Z 602.351,A -85,B 0,C 180,E1 -12710.369,E2 -12710.369} C_VEL
LIN {X 0,Y 371.155,Z 571.103,A -85,B 0,C 180,E1 -12711.264,E2 -12711.264} C_VEL
LIN {X 0,Y 372.42,Z 556.79,A -85,B 0,C 180,E1 -12714.529,E2 -12714.529} C_VEL
LIN {X 0,Y 370.829,Z 547.577,A -85,B 0,C 180,E1 -12716.809,E2 -12716.809} C_VEL
LIN {X 0,Y 368.957,Z 538.528,A -85,B 0,C 180,E1 -12719.14,E2 -12719.14} C_VEL
LIN {X 0,Y 368.897,Z 538.53,A -85,B 0,C 180,E1 -12722.237,E2 -12722.237} C_VEL
LIN {X 0,Y 368.927,Z 538.528,A -85,B 0,C 180,E1 -12725.001,E2 -12725.001} C_VEL
LIN {X 0,Y 368.907,Z 538.529,A -85,B 0,C 180,E1 -12728.64,E2 -12728.64} C_VEL
LIN {X 0,Y 368.879,Z 538.534,A -85,B 0,C 180,E1 -12732.009,E2 -12732.009} C_VEL
LIN {X 0,Y 368.923,Z 538.53,A -85,B 0,C 180,E1 -12735.182,E2 -12735.182} C_VEL
LIN {X 0,Y 368.905,Z 538.529,A -85,B 0,C 180,E1 -12738.181,E2 -12738.181} C_VEL
LIN {X 0,Y 368.908,Z 538.534,A -85,B 0,C 180,E1 -12741.358,E2 -12741.358} C_VEL
LIN {X 0,Y 368.931,Z 538.529,A -85,B 0,C 180,E1 -12745.146,E2 -12745.146} C_VEL
LIN {X 0,Y 368.923,Z 538.529,A -85,B 0,C 180,E1 -12749.046,E2 -12749.046} C_VEL
LIN {X 0,Y 368.98,Z 538.525,A -85,B 0,C 180,E1 -12751.564,E2 -12751.564} C_VEL
LIN {X 0,Y 368.993,Z 538.519,A -85,B 0,C 180,E1 -12754.019,E2 -12754.019} C_VEL
LIN {X 0,Y 368.917,Z 538.532,A -85,B 0,C 180,E1 -12757.604,E2 -12757.604} C_VEL
LIN {X 0,Y 368.974,Z 538.523,A -85,B 0,C 180,E1 -12761.107,E2 -12761.107} C_VEL
LIN {X 0,Y 368.99,Z 538.518,A -85,B 0,C 180,E1 -12764.535,E2 -12764.535} C_VEL
LIN {X 0,Y 368.997,Z 538.519,A -85,B 0,C 180,E1 -12767.907,E2 -12767.907} C_VEL
LIN {X 0,Y 369.181,Z 538.497,A -85,B 0,C 180,E1 -12771.844,E2 -12771.844} C_VEL
LIN {X 0,Y 369.136,Z 538.5,A -85,B 0,C 180,E1 -12774.538,E2 -12774.538} C_VEL
LIN {X 0,Y 369.31,Z 538.481,A -85,B 0,C 180,E1 -12777.819,E2 -12777.819} C_VEL
LIN {X 0,Y 369.449,Z 538.462,A -85,B 0,C 180,E1 -12780,E2 -12780} C_VEL
LIN {X 0,Y 369.311,Z 538.479,A -85,B 0,C 180,E1 -12782.181,E2 -12782.181} C_VEL
LIN {X 0,Y 369.19,Z 538.493,A -85,B 0,C 180,E1 -12786.604,E2 -12786.604} C_VEL
LIN {X 0,Y 369.06,Z 538.512,A -85,B 0,C 180,E1 -12789.869,E2 -12789.869} C_VEL
LIN {X 0,Y 369.029,Z 538.516,A -85,B 0,C 180,E1 -12793.773,E2 -12793.773} C_VEL
LIN {X 0,Y 368.994,Z 538.521,A -85,B 0,C 180,E1 -12797.769,E2 -12797.769} C_VEL
LIN {X 0,Y 368.923,Z 538.531,A -85,B 0,C 180,E1 -12801.22,E2 -12801.22} C_VEL
LIN {X 0,Y 368.951,Z 538.524,A -85,B 0,C 180,E1 -12804.776,E2 -12804.776} C_VEL
LIN {X 0,Y 368.981,Z 538.519,A -85,B 0,C 180,E1 -12808.436,E2 -12808.436} C_VEL
LIN {X 0,Y 368.894,Z 538.53,A -85,B 0,C 180,E1 -12812.239,E2 -12812.239} C_VEL
LIN {X 0,Y 368.924,Z 538.529,A -85,B 0,C 180,E1 -12815.002,E2 -12815.002} C_VEL
LIN {X 0,Y 368.906,Z 538.529,A -85,B 0,C 180,E1 -12818.642,E2 -12818.642} C_VEL
LIN {X 0,Y 368.879,Z 538.533,A -85,B 0,C 180,E1 -12822.01,E2 -12822.01} C_VEL
LIN {X 0,Y 368.952,Z 538.527,A -85,B 0,C 180,E1 -12825.188,E2 -12825.188} C_VEL
LIN {X 0,Y 368.939,Z 538.525,A -85,B 0,C 180,E1 -12828.187,E2 -12828.187} C_VEL
LIN {X 0,Y 368.913,Z 538.534,A -85,B 0,C 180,E1 -12831.36,E2 -12831.36} C_VEL
LIN {X 0,Y 368.936,Z 538.529,A -85,B 0,C 180,E1 -12835.147,E2 -12835.147} C_VEL
LIN {X 0,Y 368.929,Z 538.529,A -85,B 0,C 180,E1 -12839.047,E2 -12839.047} C_VEL
LIN {X 0,Y 368.981,Z 538.524,A -85,B 0,C 180,E1 -12841.565,E2 -12841.565} C_VEL
LIN {X 0,Y 369.001,Z 538.518,A -85,B 0,C 180,E1 -12844.021,E2 -12844.021} C_VEL
LIN {X 0,Y 368.935,Z 538.532,A -85,B 0,C 180,E1 -12847.606,E2 -12847.606} C_VEL
LIN {X 0,Y 368.93,Z 538.565,A -85,B 0,C 180,E1 -12849.041,E2 -12849.041} C_VEL
LIN {X 0,Y 370.93,Z 548.569,A -85,B 0,C 180,E1 -12851.915,E2 -12851.915} C_VEL
LIN {X 0,Y 371.455,Z 551.872,A -85,B 0,C 180,E1 -12852.832,E2 -12852.832} C_VEL
LIN {X 0,Y 376.381,Z 576.568,A -85,B 0,C 180,E1 -12853.596,E2 -12853.596} C_VEL
LIN {X 0,Y 375.199,Z 658.594,A -85,B 0,C 180,E1 -12855.179,E2 -12855.179} C_VEL
LIN {X 0,Y 374.717,Z 671.067,A -85,B 0,C 180,E1 -12855.611,E2 -12855.611} C_VEL
LIN {X 0,Y 374.048,Z 683.935,A -85,B 0,C 180,E1 -12856.278,E2 -12856.278} C_VEL
LIN {X 0,Y 373.219,Z 695.359,A -85,B 0,C 180,E1 -12857.079,E2 -12857.079} C_VEL
LIN {X 0,Y 372.358,Z 707.051,A -85,B 0,C 180,E1 -12858.156,E2 -12858.156} C_VEL
LIN {X 0,Y 371.279,Z 717.541,A -85,B 0,C 180,E1 -12859.365,E2 -12859.365} C_VEL
LIN {X 0,Y 370.488,Z 725.884,A -85,B 0,C 180,E1 -12860.549,E2 -12860.549} C_VEL
LIN {X 0,Y 369.708,Z 734.727,A -85,B 0,C 180,E1 -12862.079,E2 -12862.079} C_VEL
LIN {X 0,Y 368.98,Z 742.292,A -85,B 0,C 180,E1 -12863.712,E2 -12863.712} C_VEL
LIN {X 0,Y 368.543,Z 747.477,A -85,B 0,C 180,E1 -12865.077,E2 -12865.077} C_VEL
LIN {X 0,Y 367.992,Z 752.507,A -85,B 0,C 180,E1 -12866.716,E2 -12866.716} C_VEL
LIN {X 0,Y 367.701,Z 756.413,A -85,B 0,C 180,E1 -12868.357,E2 -12868.357} C_VEL
LIN {X 0,Y 367.517,Z 759.3,A -85,B 0,C 180,E1 -12870,E2 -12870} C_VEL
LIN {X 0,Y 367.471,Z 760.669,A -85,B 0,C 180,E1 -12871.096,E2 -12871.096} C_VEL
LIN {X 0,Y 367.39,Z 762.244,A -85,B 0,C 180,E1 -12873.29,E2 -12873.29} C_VEL
LIN {X 0,Y 367.428,Z 762.449,A -85,B 0,C 180,E1 -12874.388,E2 -12874.388} C_VEL
LIN {X 0,Y 367.481,Z 761.621,A -85,B 0,C 180,E1 -12876.589,E2 -12876.589} C_VEL
LIN {X 0,Y 367.537,Z 760.63,A -85,B 0,C 180,E1 -12877.692,E2 -12877.692} C_VEL
LIN {X 0,Y 367.634,Z 759.233,A -85,B 0,C 180,E1 -12878.797,E2 -12878.797} C_VEL
LIN {X 0,Y 367.851,Z 756.306,A -85,B 0,C 180,E1 -12880.457,E2 -12880.457} C_VEL
LIN {X 0,Y 368.322,Z 752.331,A -85,B 0,C 180,E1 -12882.116,E2 -12882.116} C_VEL
LIN {X 0,Y 368.872,Z 746.938,A -85,B 0,C 180,E1 -12883.848,E2 -12883.848} C_VEL
LIN {X 0,Y 369.744,Z 739.464,A -85,B 0,C 180,E1 -12885.715,E2 -12885.715} C_VEL
LIN {X 0,Y 370.78,Z 731.098,A -85,B 0,C 180,E1 -12887.369,E2 -12887.369} C_VEL
LIN {X 0,Y 371.776,Z 722.446,A -85,B 0,C 180,E1 -12888.745,E2 -12888.745} C_VEL
LIN {X 0,Y 372.901,Z 711.761,A -85,B 0,C 180,E1 -12890.117,E2 -12890.117} C_VEL
LIN {X 0,Y 373.915,Z 702.008,A -85,B 0,C 180,E1 -12891.122,E2 -12891.122} C_VEL
LIN {X 0,Y 373.766,Z 696.995,A -85,B 0,C 180,E1 -12891.608,E2 -12891.608} C_VEL
LIN {X 0,Y 371.641,Z 688.761,A -85,B 0,C 180,E1 -12892.41,E2 -12892.41} C_VEL
LIN {X 0,Y 369.512,Z 680.177,A -85,B 0,C 180,E1 -12893.101,E2 -12893.101} C_VEL
LIN {X 0,Y 369.331,Z 674.63,A -85,B 0,C 180,E1 -12893.406,E2 -12893.406} C_VEL
LIN {X 0,Y 369.975,Z 661.65,A -85,B 0,C 180,E1 -12893.907,E2 -12893.907} C_VEL
